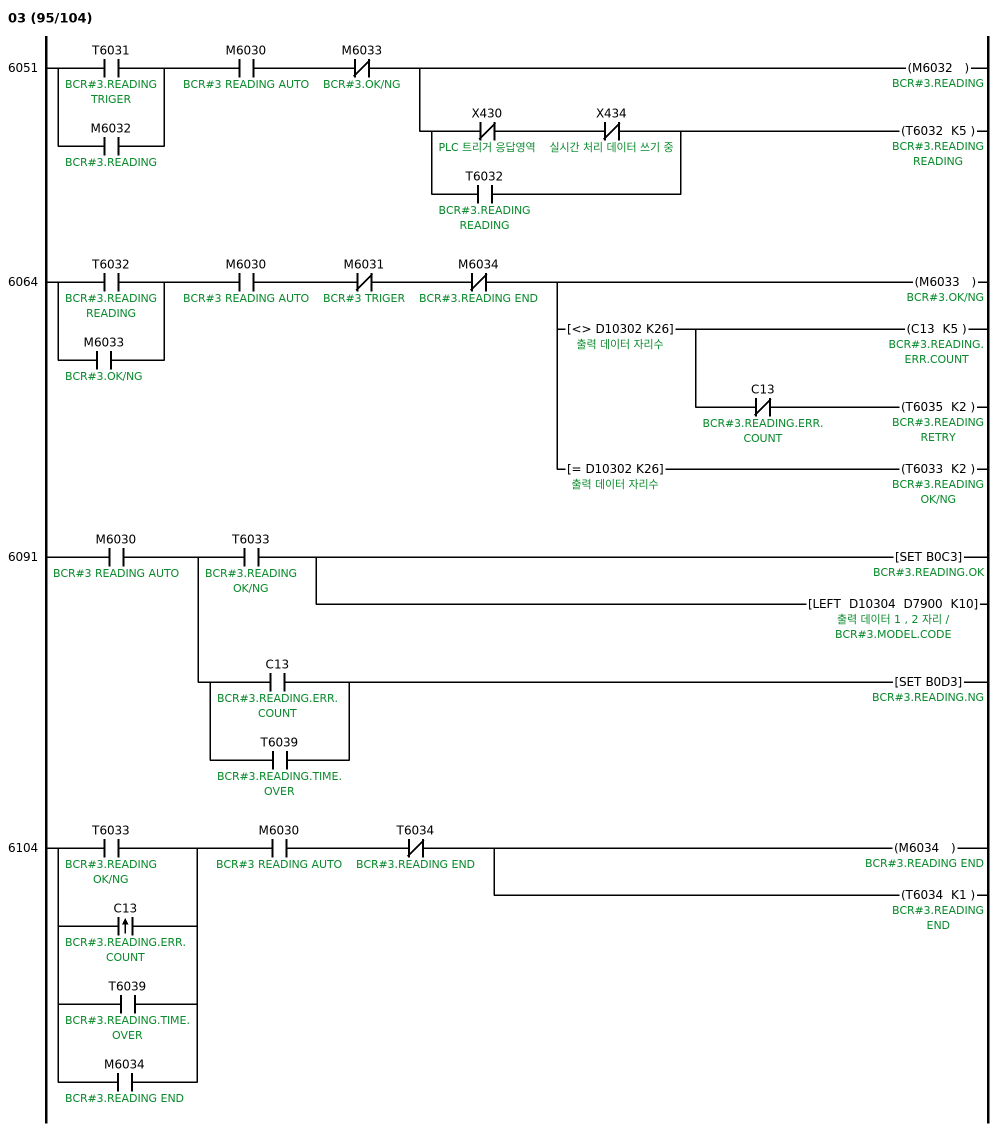
6051  LD      T6031  ; BCR#3.READING TRIGER
      OR      M6032  ; BCR#3.READING
      AND     M6030  ; BCR#3 READING AUTO
      ANI     M6033  ; BCR#3.OK/NG
      OUT     M6032  ; BCR#3.READING
      LDI     X430  ; PLC 트리거 응답영역
      ANI     X434  ; 실시간 처리 데이터 쓰기 중
      OR      T6032  ; BCR#3.READING READING
      ANB
      OUT     T6032 K5  ; BCR#3.READING READING
6064  LD      T6032  ; BCR#3.READING READING
      OR      M6033  ; BCR#3.OK/NG
      AND     M6030  ; BCR#3 READING AUTO
      ANI     M6031  ; BCR#3 TRIGER
      ANI     M6034  ; BCR#3.READING END
      OUT     M6033  ; BCR#3.OK/NG
      MPS
      AND<>   D10302 K26  ; 출력 데이터 자리수
      OUT     C13 K5  ; BCR#3.READING.ERR.COUNT
      ANI     C13  ; BCR#3.READING.ERR.COUNT
      OUT     T6035 K2  ; BCR#3.READING RETRY
      MPP
      AND=    D10302 K26  ; 출력 데이터 자리수
      OUT     T6033 K2  ; BCR#3.READING OK/NG
6091  LD      M6030  ; BCR#3 READING AUTO
      MPS
      AND     T6033  ; BCR#3.READING OK/NG
      SET     B0C3  ; BCR#3.READING.OK
      LEFT    D10304 D7900 K10  ; BCR#3.MODEL.CODE
      MPP
      LD      C13  ; BCR#3.READING.ERR.COUNT
      OR      T6039  ; BCR#3.READING.TIME.OVER
      ANB
      SET     B0D3  ; BCR#3.READING.NG
6104  LD      T6033  ; BCR#3.READING OK/NG
      ORP     C13  ; BCR#3.READING.ERR.COUNT
      OR      T6039  ; BCR#3.READING.TIME.OVER
      OR      M6034  ; BCR#3.READING END
      AND     M6030  ; BCR#3 READING AUTO
      ANI     T6034  ; BCR#3.READING END
      OUT     M6034  ; BCR#3.READING END
      OUT     T6034 K1  ; BCR#3.READING END
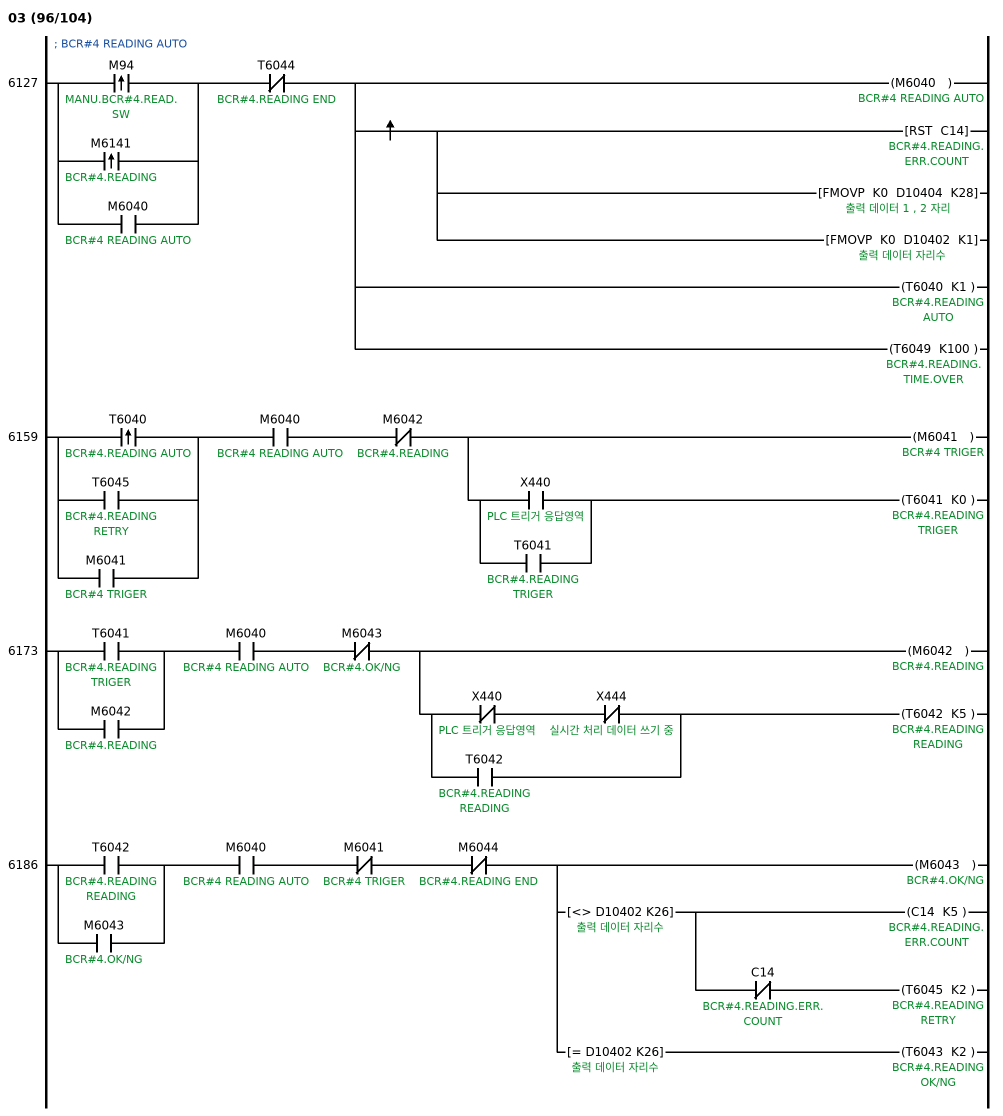
; BCR#4 READING AUTO
6127  LDP     M94  ; MANU.BCR#4.READ.SW
      ORP     M6141  ; BCR#4.READING
      OR      M6040  ; BCR#4 READING AUTO
      ANI     T6044  ; BCR#4.READING END
      OUT     M6040  ; BCR#4 READING AUTO
      MPS
      MEP
      RST     C14  ; BCR#4.READING.ERR.COUNT
      FMOVP   K0 D10404 K28  ; 출력 데이터 1 , 2 자리
      FMOVP   K0 D10402 K1  ; 출력 데이터 자리수
      MPP
      OUT     T6040 K1  ; BCR#4.READING AUTO
      OUT     T6049 K100  ; BCR#4.READING.TIME.OVER
6159  LDP     T6040  ; BCR#4.READING AUTO
      OR      T6045  ; BCR#4.READING RETRY
      OR      M6041  ; BCR#4 TRIGER
      AND     M6040  ; BCR#4 READING AUTO
      ANI     M6042  ; BCR#4.READING
      OUT     M6041  ; BCR#4 TRIGER
      LD      X440  ; PLC 트리거 응답영역
      OR      T6041  ; BCR#4.READING TRIGER
      ANB
      OUT     T6041 K0  ; BCR#4.READING TRIGER
6173  LD      T6041  ; BCR#4.READING TRIGER
      OR      M6042  ; BCR#4.READING
      AND     M6040  ; BCR#4 READING AUTO
      ANI     M6043  ; BCR#4.OK/NG
      OUT     M6042  ; BCR#4.READING
      LDI     X440  ; PLC 트리거 응답영역
      ANI     X444  ; 실시간 처리 데이터 쓰기 중
      OR      T6042  ; BCR#4.READING READING
      ANB
      OUT     T6042 K5  ; BCR#4.READING READING
6186  LD      T6042  ; BCR#4.READING READING
      OR      M6043  ; BCR#4.OK/NG
      AND     M6040  ; BCR#4 READING AUTO
      ANI     M6041  ; BCR#4 TRIGER
      ANI     M6044  ; BCR#4.READING END
      OUT     M6043  ; BCR#4.OK/NG
      MPS
      AND<>   D10402 K26  ; 출력 데이터 자리수
      OUT     C14 K5  ; BCR#4.READING.ERR.COUNT
      ANI     C14  ; BCR#4.READING.ERR.COUNT
      OUT     T6045 K2  ; BCR#4.READING RETRY
      MPP
      AND=    D10402 K26  ; 출력 데이터 자리수
      OUT     T6043 K2  ; BCR#4.READING OK/NG
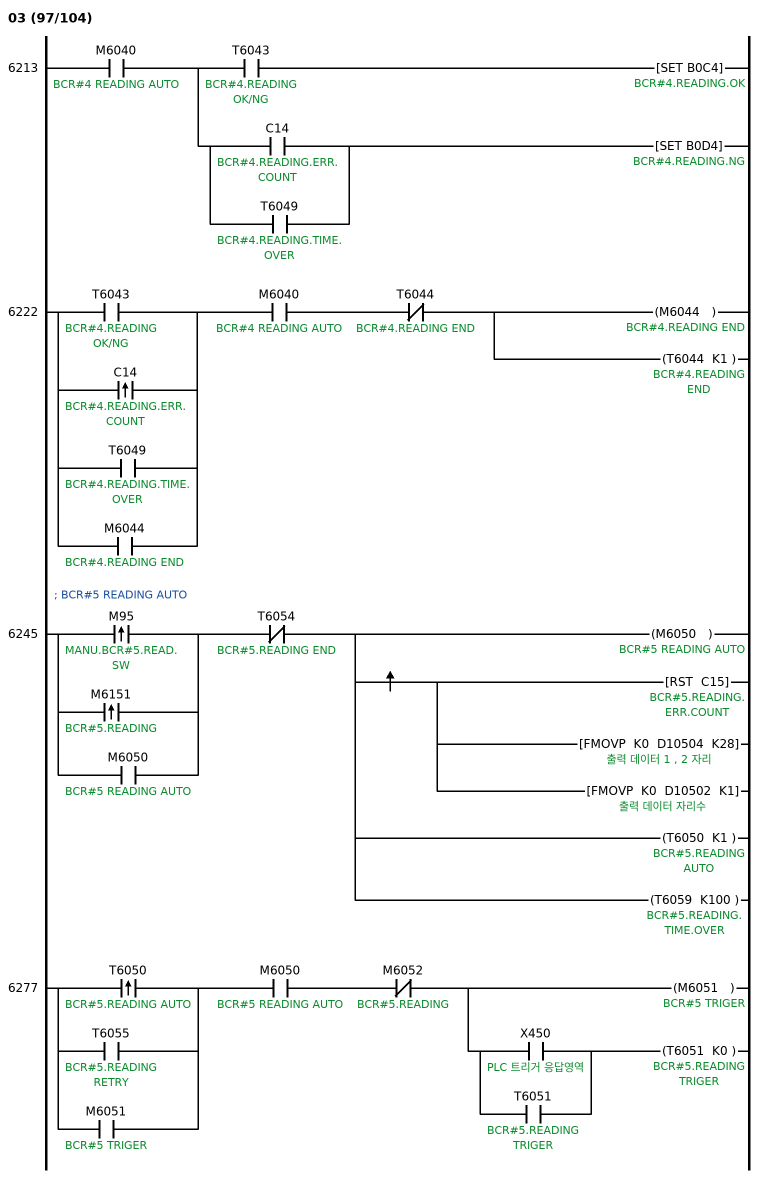
6213  LD      M6040  ; BCR#4 READING AUTO
      MPS
      AND     T6043  ; BCR#4.READING OK/NG
      SET     B0C4  ; BCR#4.READING.OK
      MPP
      LD      C14  ; BCR#4.READING.ERR.COUNT
      OR      T6049  ; BCR#4.READING.TIME.OVER
      ANB
      SET     B0D4  ; BCR#4.READING.NG
6222  LD      T6043  ; BCR#4.READING OK/NG
      ORP     C14  ; BCR#4.READING.ERR.COUNT
      OR      T6049  ; BCR#4.READING.TIME.OVER
      OR      M6044  ; BCR#4.READING END
      AND     M6040  ; BCR#4 READING AUTO
      ANI     T6044  ; BCR#4.READING END
      OUT     M6044  ; BCR#4.READING END
      OUT     T6044 K1  ; BCR#4.READING END
; BCR#5 READING AUTO
6245  LDP     M95  ; MANU.BCR#5.READ.SW
      ORP     M6151  ; BCR#5.READING
      OR      M6050  ; BCR#5 READING AUTO
      ANI     T6054  ; BCR#5.READING END
      OUT     M6050  ; BCR#5 READING AUTO
      MPS
      MEP
      RST     C15  ; BCR#5.READING.ERR.COUNT
      FMOVP   K0 D10504 K28  ; 출력 데이터 1 , 2 자리
      FMOVP   K0 D10502 K1  ; 출력 데이터 자리수
      MPP
      OUT     T6050 K1  ; BCR#5.READING AUTO
      OUT     T6059 K100  ; BCR#5.READING.TIME.OVER
6277  LDP     T6050  ; BCR#5.READING AUTO
      OR      T6055  ; BCR#5.READING RETRY
      OR      M6051  ; BCR#5 TRIGER
      AND     M6050  ; BCR#5 READING AUTO
      ANI     M6052  ; BCR#5.READING
      OUT     M6051  ; BCR#5 TRIGER
      LD      X450  ; PLC 트리거 응답영역
      OR      T6051  ; BCR#5.READING TRIGER
      ANB
      OUT     T6051 K0  ; BCR#5.READING TRIGER
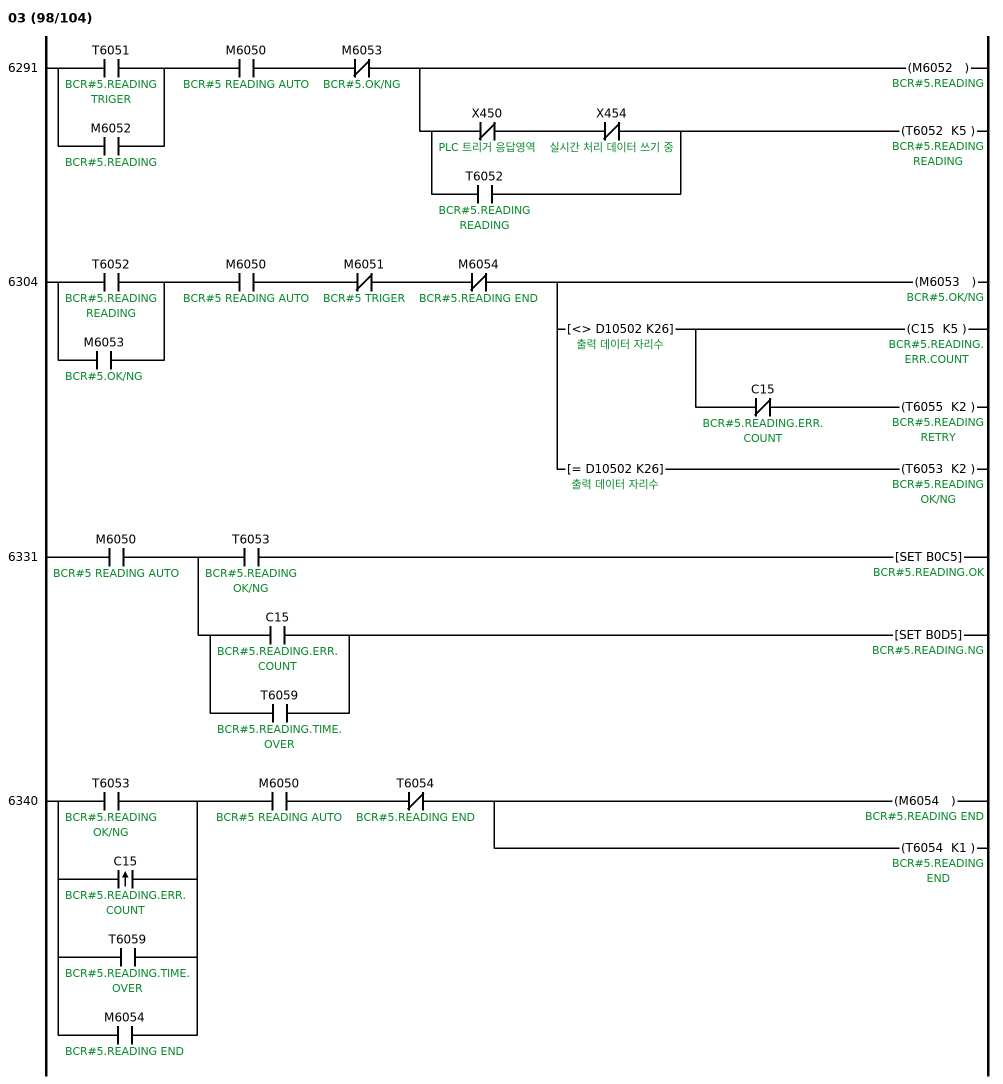
6291  LD      T6051  ; BCR#5.READING TRIGER
      OR      M6052  ; BCR#5.READING
      AND     M6050  ; BCR#5 READING AUTO
      ANI     M6053  ; BCR#5.OK/NG
      OUT     M6052  ; BCR#5.READING
      LDI     X450  ; PLC 트리거 응답영역
      ANI     X454  ; 실시간 처리 데이터 쓰기 중
      OR      T6052  ; BCR#5.READING READING
      ANB
      OUT     T6052 K5  ; BCR#5.READING READING
6304  LD      T6052  ; BCR#5.READING READING
      OR      M6053  ; BCR#5.OK/NG
      AND     M6050  ; BCR#5 READING AUTO
      ANI     M6051  ; BCR#5 TRIGER
      ANI     M6054  ; BCR#5.READING END
      OUT     M6053  ; BCR#5.OK/NG
      MPS
      AND<>   D10502 K26  ; 출력 데이터 자리수
      OUT     C15 K5  ; BCR#5.READING.ERR.COUNT
      ANI     C15  ; BCR#5.READING.ERR.COUNT
      OUT     T6055 K2  ; BCR#5.READING RETRY
      MPP
      AND=    D10502 K26  ; 출력 데이터 자리수
      OUT     T6053 K2  ; BCR#5.READING OK/NG
6331  LD      M6050  ; BCR#5 READING AUTO
      MPS
      AND     T6053  ; BCR#5.READING OK/NG
      SET     B0C5  ; BCR#5.READING.OK
      MPP
      LD      C15  ; BCR#5.READING.ERR.COUNT
      OR      T6059  ; BCR#5.READING.TIME.OVER
      ANB
      SET     B0D5  ; BCR#5.READING.NG
6340  LD      T6053  ; BCR#5.READING OK/NG
      ORP     C15  ; BCR#5.READING.ERR.COUNT
      OR      T6059  ; BCR#5.READING.TIME.OVER
      OR      M6054  ; BCR#5.READING END
      AND     M6050  ; BCR#5 READING AUTO
      ANI     T6054  ; BCR#5.READING END
      OUT     M6054  ; BCR#5.READING END
      OUT     T6054 K1  ; BCR#5.READING END
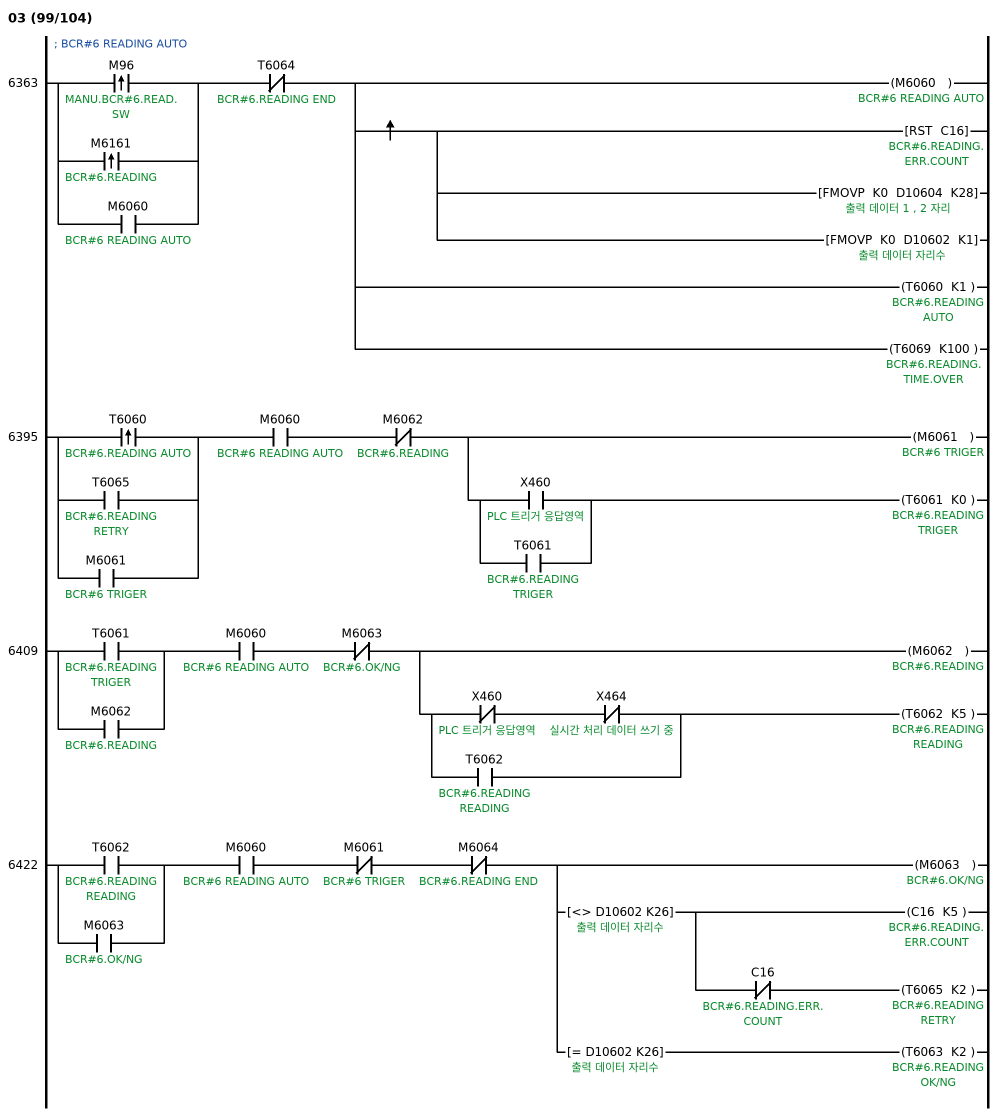
; BCR#6 READING AUTO
6363  LDP     M96  ; MANU.BCR#6.READ.SW
      ORP     M6161  ; BCR#6.READING
      OR      M6060  ; BCR#6 READING AUTO
      ANI     T6064  ; BCR#6.READING END
      OUT     M6060  ; BCR#6 READING AUTO
      MPS
      MEP
      RST     C16  ; BCR#6.READING.ERR.COUNT
      FMOVP   K0 D10604 K28  ; 출력 데이터 1 , 2 자리
      FMOVP   K0 D10602 K1  ; 출력 데이터 자리수
      MPP
      OUT     T6060 K1  ; BCR#6.READING AUTO
      OUT     T6069 K100  ; BCR#6.READING.TIME.OVER
6395  LDP     T6060  ; BCR#6.READING AUTO
      OR      T6065  ; BCR#6.READING RETRY
      OR      M6061  ; BCR#6 TRIGER
      AND     M6060  ; BCR#6 READING AUTO
      ANI     M6062  ; BCR#6.READING
      OUT     M6061  ; BCR#6 TRIGER
      LD      X460  ; PLC 트리거 응답영역
      OR      T6061  ; BCR#6.READING TRIGER
      ANB
      OUT     T6061 K0  ; BCR#6.READING TRIGER
6409  LD      T6061  ; BCR#6.READING TRIGER
      OR      M6062  ; BCR#6.READING
      AND     M6060  ; BCR#6 READING AUTO
      ANI     M6063  ; BCR#6.OK/NG
      OUT     M6062  ; BCR#6.READING
      LDI     X460  ; PLC 트리거 응답영역
      ANI     X464  ; 실시간 처리 데이터 쓰기 중
      OR      T6062  ; BCR#6.READING READING
      ANB
      OUT     T6062 K5  ; BCR#6.READING READING
6422  LD      T6062  ; BCR#6.READING READING
      OR      M6063  ; BCR#6.OK/NG
      AND     M6060  ; BCR#6 READING AUTO
      ANI     M6061  ; BCR#6 TRIGER
      ANI     M6064  ; BCR#6.READING END
      OUT     M6063  ; BCR#6.OK/NG
      MPS
      AND<>   D10602 K26  ; 출력 데이터 자리수
      OUT     C16 K5  ; BCR#6.READING.ERR.COUNT
      ANI     C16  ; BCR#6.READING.ERR.COUNT
      OUT     T6065 K2  ; BCR#6.READING RETRY
      MPP
      AND=    D10602 K26  ; 출력 데이터 자리수
      OUT     T6063 K2  ; BCR#6.READING OK/NG
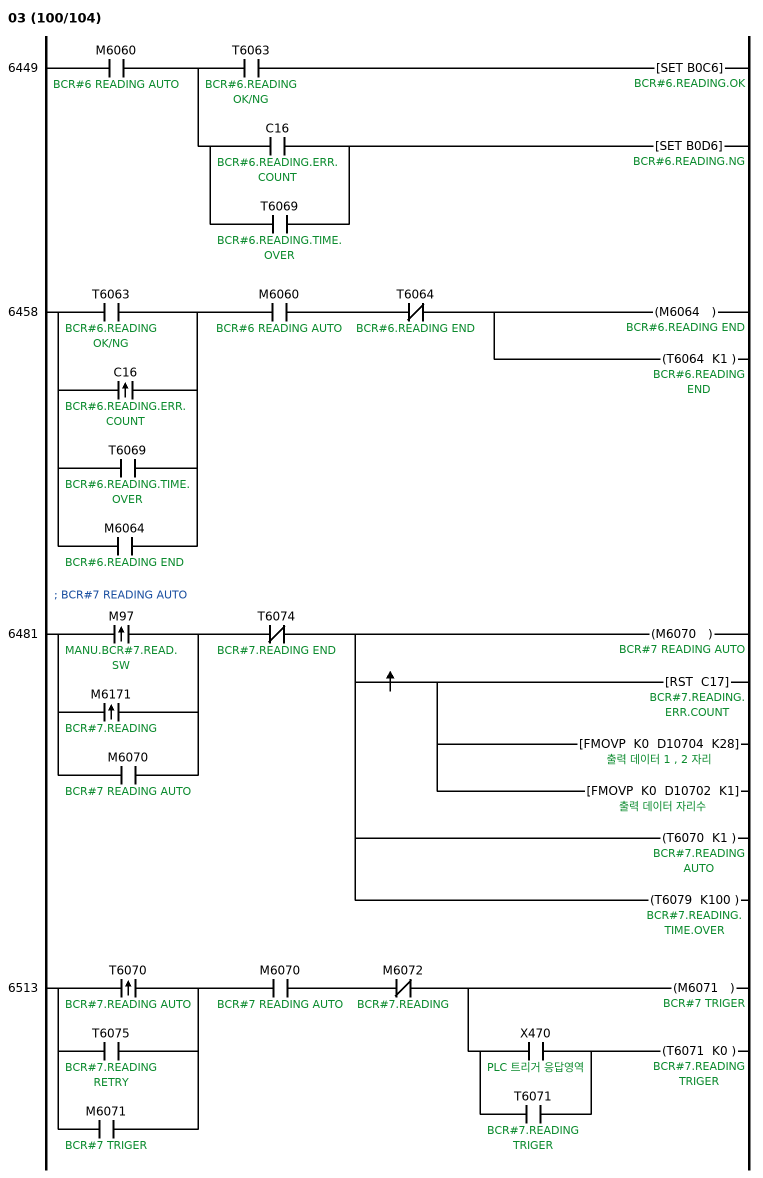
6449  LD      M6060  ; BCR#6 READING AUTO
      MPS
      AND     T6063  ; BCR#6.READING OK/NG
      SET     B0C6  ; BCR#6.READING.OK
      MPP
      LD      C16  ; BCR#6.READING.ERR.COUNT
      OR      T6069  ; BCR#6.READING.TIME.OVER
      ANB
      SET     B0D6  ; BCR#6.READING.NG
6458  LD      T6063  ; BCR#6.READING OK/NG
      ORP     C16  ; BCR#6.READING.ERR.COUNT
      OR      T6069  ; BCR#6.READING.TIME.OVER
      OR      M6064  ; BCR#6.READING END
      AND     M6060  ; BCR#6 READING AUTO
      ANI     T6064  ; BCR#6.READING END
      OUT     M6064  ; BCR#6.READING END
      OUT     T6064 K1  ; BCR#6.READING END
; BCR#7 READING AUTO
6481  LDP     M97  ; MANU.BCR#7.READ.SW
      ORP     M6171  ; BCR#7.READING
      OR      M6070  ; BCR#7 READING AUTO
      ANI     T6074  ; BCR#7.READING END
      OUT     M6070  ; BCR#7 READING AUTO
      MPS
      MEP
      RST     C17  ; BCR#7.READING.ERR.COUNT
      FMOVP   K0 D10704 K28  ; 출력 데이터 1 , 2 자리
      FMOVP   K0 D10702 K1  ; 출력 데이터 자리수
      MPP
      OUT     T6070 K1  ; BCR#7.READING AUTO
      OUT     T6079 K100  ; BCR#7.READING.TIME.OVER
6513  LDP     T6070  ; BCR#7.READING AUTO
      OR      T6075  ; BCR#7.READING RETRY
      OR      M6071  ; BCR#7 TRIGER
      AND     M6070  ; BCR#7 READING AUTO
      ANI     M6072  ; BCR#7.READING
      OUT     M6071  ; BCR#7 TRIGER
      LD      X470  ; PLC 트리거 응답영역
      OR      T6071  ; BCR#7.READING TRIGER
      ANB
      OUT     T6071 K0  ; BCR#7.READING TRIGER
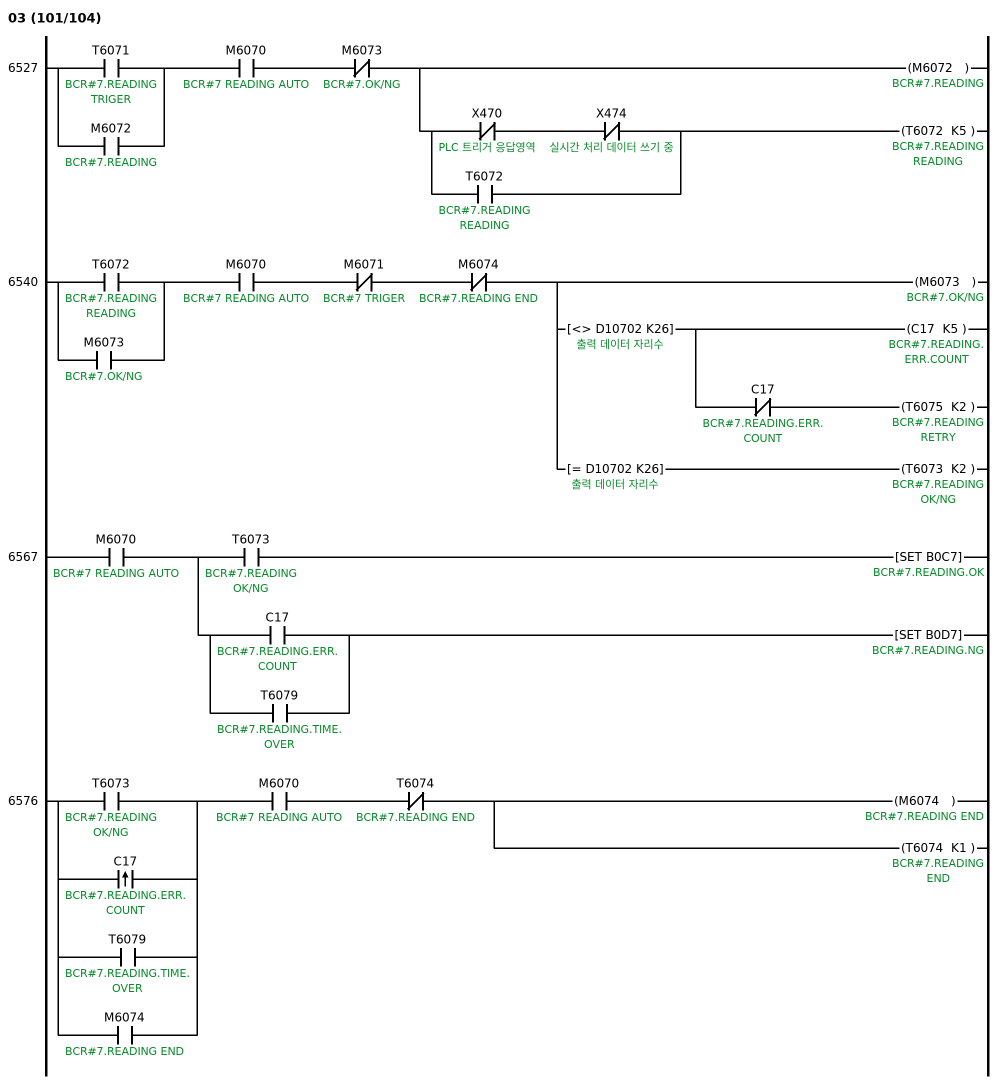
6527  LD      T6071  ; BCR#7.READING TRIGER
      OR      M6072  ; BCR#7.READING
      AND     M6070  ; BCR#7 READING AUTO
      ANI     M6073  ; BCR#7.OK/NG
      OUT     M6072  ; BCR#7.READING
      LDI     X470  ; PLC 트리거 응답영역
      ANI     X474  ; 실시간 처리 데이터 쓰기 중
      OR      T6072  ; BCR#7.READING READING
      ANB
      OUT     T6072 K5  ; BCR#7.READING READING
6540  LD      T6072  ; BCR#7.READING READING
      OR      M6073  ; BCR#7.OK/NG
      AND     M6070  ; BCR#7 READING AUTO
      ANI     M6071  ; BCR#7 TRIGER
      ANI     M6074  ; BCR#7.READING END
      OUT     M6073  ; BCR#7.OK/NG
      MPS
      AND<>   D10702 K26  ; 출력 데이터 자리수
      OUT     C17 K5  ; BCR#7.READING.ERR.COUNT
      ANI     C17  ; BCR#7.READING.ERR.COUNT
      OUT     T6075 K2  ; BCR#7.READING RETRY
      MPP
      AND=    D10702 K26  ; 출력 데이터 자리수
      OUT     T6073 K2  ; BCR#7.READING OK/NG
6567  LD      M6070  ; BCR#7 READING AUTO
      MPS
      AND     T6073  ; BCR#7.READING OK/NG
      SET     B0C7  ; BCR#7.READING.OK
      MPP
      LD      C17  ; BCR#7.READING.ERR.COUNT
      OR      T6079  ; BCR#7.READING.TIME.OVER
      ANB
      SET     B0D7  ; BCR#7.READING.NG
6576  LD      T6073  ; BCR#7.READING OK/NG
      ORP     C17  ; BCR#7.READING.ERR.COUNT
      OR      T6079  ; BCR#7.READING.TIME.OVER
      OR      M6074  ; BCR#7.READING END
      AND     M6070  ; BCR#7 READING AUTO
      ANI     T6074  ; BCR#7.READING END
      OUT     M6074  ; BCR#7.READING END
      OUT     T6074 K1  ; BCR#7.READING END
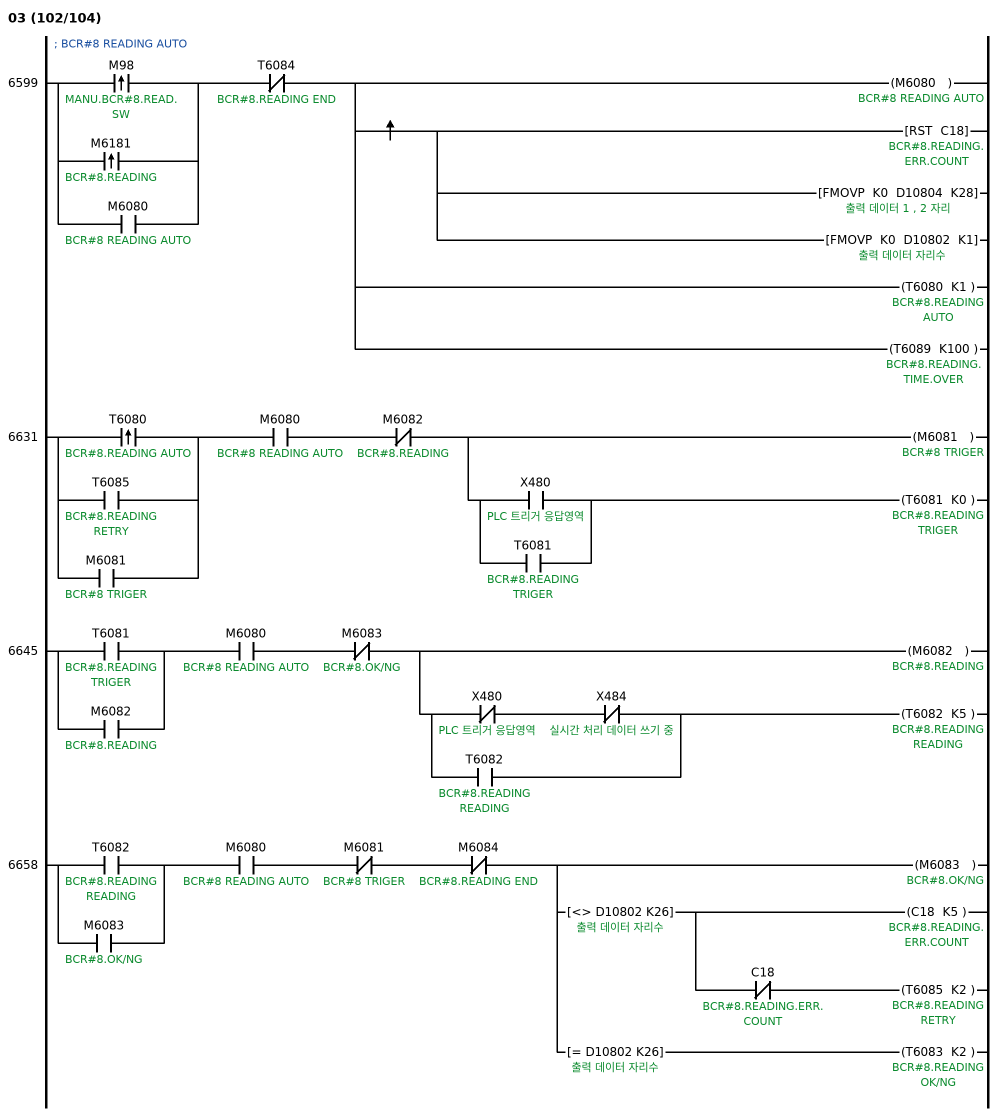
; BCR#8 READING AUTO
6599  LDP     M98  ; MANU.BCR#8.READ.SW
      ORP     M6181  ; BCR#8.READING
      OR      M6080  ; BCR#8 READING AUTO
      ANI     T6084  ; BCR#8.READING END
      OUT     M6080  ; BCR#8 READING AUTO
      MPS
      MEP
      RST     C18  ; BCR#8.READING.ERR.COUNT
      FMOVP   K0 D10804 K28  ; 출력 데이터 1 , 2 자리
      FMOVP   K0 D10802 K1  ; 출력 데이터 자리수
      MPP
      OUT     T6080 K1  ; BCR#8.READING AUTO
      OUT     T6089 K100  ; BCR#8.READING.TIME.OVER
6631  LDP     T6080  ; BCR#8.READING AUTO
      OR      T6085  ; BCR#8.READING RETRY
      OR      M6081  ; BCR#8 TRIGER
      AND     M6080  ; BCR#8 READING AUTO
      ANI     M6082  ; BCR#8.READING
      OUT     M6081  ; BCR#8 TRIGER
      LD      X480  ; PLC 트리거 응답영역
      OR      T6081  ; BCR#8.READING TRIGER
      ANB
      OUT     T6081 K0  ; BCR#8.READING TRIGER
6645  LD      T6081  ; BCR#8.READING TRIGER
      OR      M6082  ; BCR#8.READING
      AND     M6080  ; BCR#8 READING AUTO
      ANI     M6083  ; BCR#8.OK/NG
      OUT     M6082  ; BCR#8.READING
      LDI     X480  ; PLC 트리거 응답영역
      ANI     X484  ; 실시간 처리 데이터 쓰기 중
      OR      T6082  ; BCR#8.READING READING
      ANB
      OUT     T6082 K5  ; BCR#8.READING READING
6658  LD      T6082  ; BCR#8.READING READING
      OR      M6083  ; BCR#8.OK/NG
      AND     M6080  ; BCR#8 READING AUTO
      ANI     M6081  ; BCR#8 TRIGER
      ANI     M6084  ; BCR#8.READING END
      OUT     M6083  ; BCR#8.OK/NG
      MPS
      AND<>   D10802 K26  ; 출력 데이터 자리수
      OUT     C18 K5  ; BCR#8.READING.ERR.COUNT
      ANI     C18  ; BCR#8.READING.ERR.COUNT
      OUT     T6085 K2  ; BCR#8.READING RETRY
      MPP
      AND=    D10802 K26  ; 출력 데이터 자리수
      OUT     T6083 K2  ; BCR#8.READING OK/NG
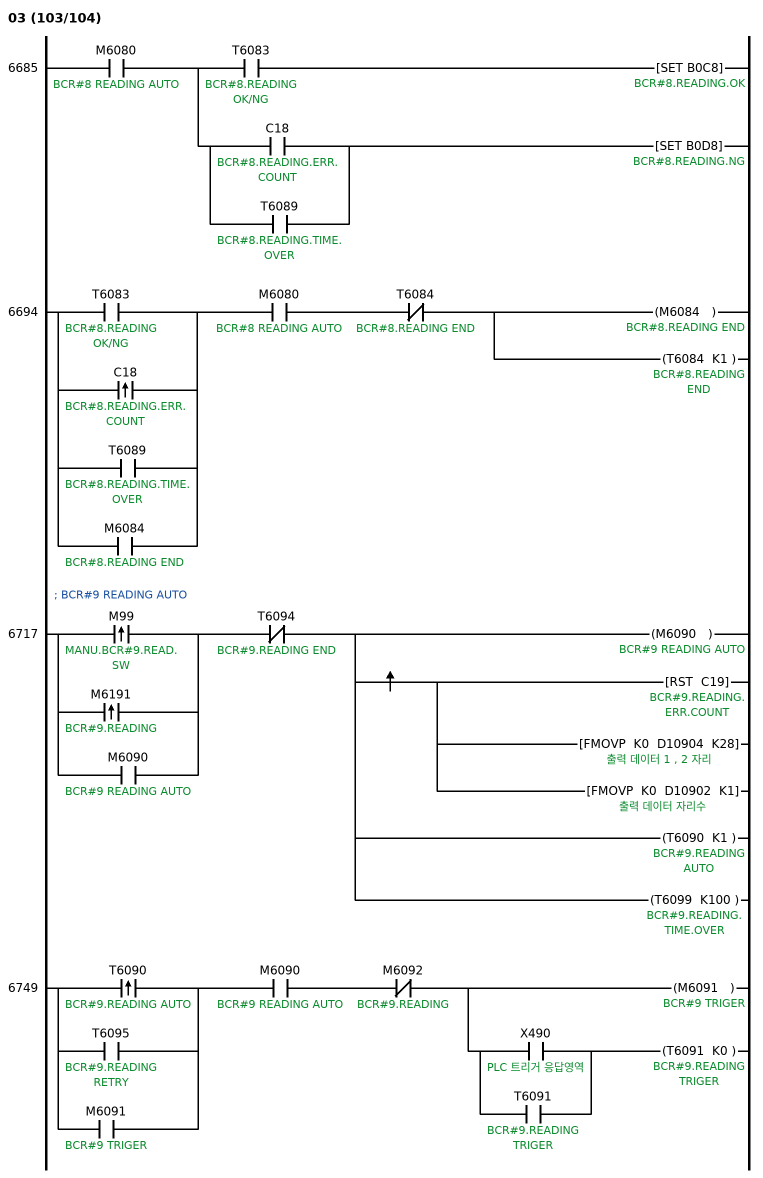
6685  LD      M6080  ; BCR#8 READING AUTO
      MPS
      AND     T6083  ; BCR#8.READING OK/NG
      SET     B0C8  ; BCR#8.READING.OK
      MPP
      LD      C18  ; BCR#8.READING.ERR.COUNT
      OR      T6089  ; BCR#8.READING.TIME.OVER
      ANB
      SET     B0D8  ; BCR#8.READING.NG
6694  LD      T6083  ; BCR#8.READING OK/NG
      ORP     C18  ; BCR#8.READING.ERR.COUNT
      OR      T6089  ; BCR#8.READING.TIME.OVER
      OR      M6084  ; BCR#8.READING END
      AND     M6080  ; BCR#8 READING AUTO
      ANI     T6084  ; BCR#8.READING END
      OUT     M6084  ; BCR#8.READING END
      OUT     T6084 K1  ; BCR#8.READING END
; BCR#9 READING AUTO
6717  LDP     M99  ; MANU.BCR#9.READ.SW
      ORP     M6191  ; BCR#9.READING
      OR      M6090  ; BCR#9 READING AUTO
      ANI     T6094  ; BCR#9.READING END
      OUT     M6090  ; BCR#9 READING AUTO
      MPS
      MEP
      RST     C19  ; BCR#9.READING.ERR.COUNT
      FMOVP   K0 D10904 K28  ; 출력 데이터 1 , 2 자리
      FMOVP   K0 D10902 K1  ; 출력 데이터 자리수
      MPP
      OUT     T6090 K1  ; BCR#9.READING AUTO
      OUT     T6099 K100  ; BCR#9.READING.TIME.OVER
6749  LDP     T6090  ; BCR#9.READING AUTO
      OR      T6095  ; BCR#9.READING RETRY
      OR      M6091  ; BCR#9 TRIGER
      AND     M6090  ; BCR#9 READING AUTO
      ANI     M6092  ; BCR#9.READING
      OUT     M6091  ; BCR#9 TRIGER
      LD      X490  ; PLC 트리거 응답영역
      OR      T6091  ; BCR#9.READING TRIGER
      ANB
      OUT     T6091 K0  ; BCR#9.READING TRIGER
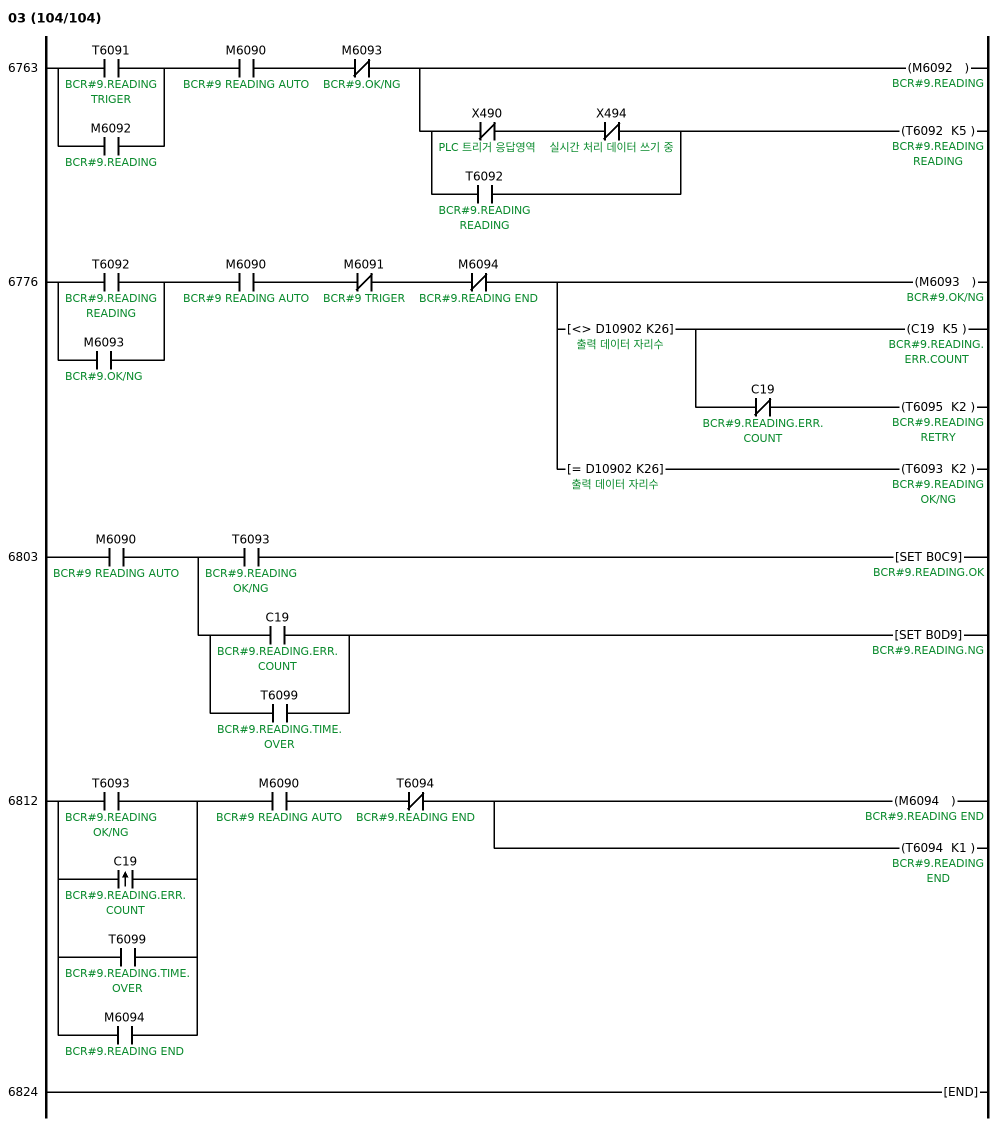
6763  LD      T6091  ; BCR#9.READING TRIGER
      OR      M6092  ; BCR#9.READING
      AND     M6090  ; BCR#9 READING AUTO
      ANI     M6093  ; BCR#9.OK/NG
      OUT     M6092  ; BCR#9.READING
      LDI     X490  ; PLC 트리거 응답영역
      ANI     X494  ; 실시간 처리 데이터 쓰기 중
      OR      T6092  ; BCR#9.READING READING
      ANB
      OUT     T6092 K5  ; BCR#9.READING READING
6776  LD      T6092  ; BCR#9.READING READING
      OR      M6093  ; BCR#9.OK/NG
      AND     M6090  ; BCR#9 READING AUTO
      ANI     M6091  ; BCR#9 TRIGER
      ANI     M6094  ; BCR#9.READING END
      OUT     M6093  ; BCR#9.OK/NG
      MPS
      AND<>   D10902 K26  ; 출력 데이터 자리수
      OUT     C19 K5  ; BCR#9.READING.ERR.COUNT
      ANI     C19  ; BCR#9.READING.ERR.COUNT
      OUT     T6095 K2  ; BCR#9.READING RETRY
      MPP
      AND=    D10902 K26  ; 출력 데이터 자리수
      OUT     T6093 K2  ; BCR#9.READING OK/NG
6803  LD      M6090  ; BCR#9 READING AUTO
      MPS
      AND     T6093  ; BCR#9.READING OK/NG
      SET     B0C9  ; BCR#9.READING.OK
      MPP
      LD      C19  ; BCR#9.READING.ERR.COUNT
      OR      T6099  ; BCR#9.READING.TIME.OVER
      ANB
      SET     B0D9  ; BCR#9.READING.NG
6812  LD      T6093  ; BCR#9.READING OK/NG
      ORP     C19  ; BCR#9.READING.ERR.COUNT
      OR      T6099  ; BCR#9.READING.TIME.OVER
      OR      M6094  ; BCR#9.READING END
      AND     M6090  ; BCR#9 READING AUTO
      ANI     T6094  ; BCR#9.READING END
      OUT     M6094  ; BCR#9.READING END
      OUT     T6094 K1  ; BCR#9.READING END
6824  END
END_PROGRAM

PROGRAM 04  // SERVO
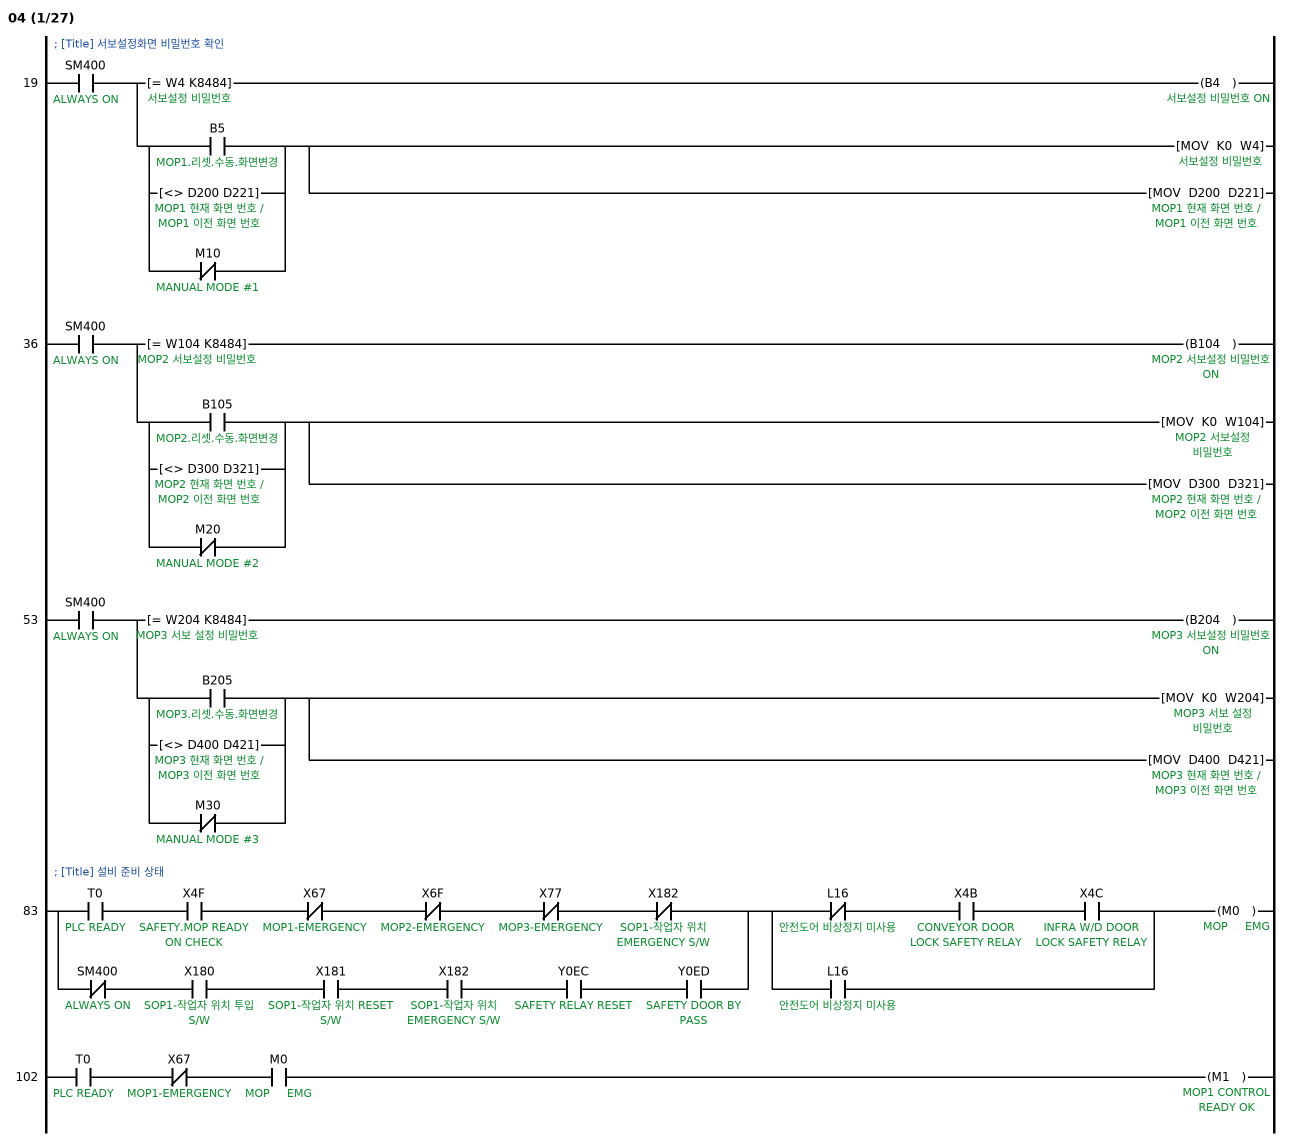
; [Title] 서보설정화면 비밀번호 확인
19    LD      SM400  ; ALWAYS ON
      MPS
      AND=    W4 K8484  ; 서보설정 비밀번호
      OUT     B4  ; 서보설정 비밀번호 ON
      MPP
      LD      B5  ; MOP1.리셋.수동.화면변경
      OR<>    D200 D221  ; MOP1 현재 화면 번호 / MOP1 이전 화면 번호
      ORI     M10  ; MANUAL MODE #1
      ANB
      MOV     K0 W4
      MOV     D200 D221
36    LD      SM400  ; ALWAYS ON
      MPS
      AND=    W104 K8484  ; MOP2 서보설정 비밀번호
      OUT     B104  ; MOP2 서보설정 비밀번호 ON
      MPP
      LD      B105  ; MOP2.리셋.수동.화면변경
      OR<>    D300 D321  ; MOP2 현재 화면 번호 / MOP2 이전 화면 번호
      ORI     M20  ; MANUAL MODE #2
      ANB
      MOV     K0 W104
      MOV     D300 D321
53    LD      SM400  ; ALWAYS ON
      MPS
      AND=    W204 K8484  ; MOP3 서보 설정 비밀번호
      OUT     B204  ; MOP3 서보설정 비밀번호 ON
      MPP
      LD      B205  ; MOP3.리셋.수동.화면변경
      OR<>    D400 D421  ; MOP3 현재 화면 번호 / MOP3 이전 화면 번호
      ORI     M30  ; MANUAL MODE #3
      ANB
      MOV     K0 W204
      MOV     D400 D421
; [Title] 설비 준비 상태
83    LD      T0  ; PLC READY
      AND     X4F  ; SAFETY.MOP READY ON CHECK
      ANI     X67  ; MOP1-EMERGENCY
      ANI     X6F  ; MOP2-EMERGENCY
      ANI     X77  ; MOP3-EMERGENCY
      ANI     X182  ; SOP1-작업자 위치 EMERGENCY S/W
      LDI     SM400  ; ALWAYS ON
      AND     X180  ; SOP1-작업자 위치 투입 S/W
      AND     X181  ; SOP1-작업자 위치 RESET S/W
      AND     X182  ; SOP1-작업자 위치 EMERGENCY S/W
      AND     Y0EC  ; SAFETY RELAY RESET
      AND     Y0ED  ; SAFETY DOOR BY PASS
      ORB
      LDI     L16  ; 안전도어 비상정지 미사용
      AND     X4B  ; CONVEYOR DOOR LOCK SAFETY RELAY
      AND     X4C  ; INFRA W/D DOOR LOCK SAFETY RELAY
      OR      L16  ; 안전도어 비상정지 미사용
      ANB
      OUT     M0  ; MOP     EMG
102   LD      T0  ; PLC READY
      ANI     X67  ; MOP1-EMERGENCY
      AND     M0  ; MOP     EMG
      OUT     M1  ; MOP1 CONTROL READY OK
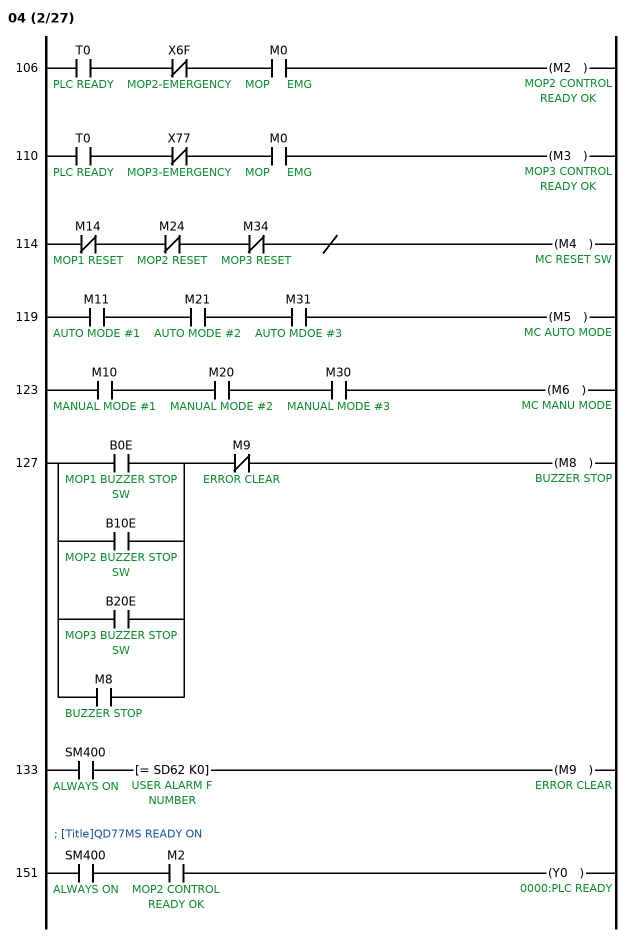
106   LD      T0  ; PLC READY
      ANI     X6F  ; MOP2-EMERGENCY
      AND     M0  ; MOP     EMG
      OUT     M2  ; MOP2 CONTROL READY OK
110   LD      T0  ; PLC READY
      ANI     X77  ; MOP3-EMERGENCY
      AND     M0  ; MOP     EMG
      OUT     M3  ; MOP3 CONTROL READY OK
114   LDI     M14  ; MOP1 RESET
      ANI     M24  ; MOP2 RESET
      ANI     M34  ; MOP3 RESET
      INV
      OUT     M4  ; MC RESET SW
119   LD      M11  ; AUTO MODE #1
      AND     M21  ; AUTO MODE #2
      AND     M31  ; AUTO MDOE #3
      OUT     M5  ; MC AUTO MODE
123   LD      M10  ; MANUAL MODE #1
      AND     M20  ; MANUAL MODE #2
      AND     M30  ; MANUAL MODE #3
      OUT     M6  ; MC MANU MODE
127   LD      B0E  ; MOP1 BUZZER STOP SW
      OR      B10E  ; MOP2 BUZZER STOP SW
      OR      B20E  ; MOP3 BUZZER STOP SW
      OR      M8  ; BUZZER STOP
      ANI     M9  ; ERROR CLEAR
      OUT     M8  ; BUZZER STOP
133   LD      SM400  ; ALWAYS ON
      AND=    SD62 K0  ; USER ALARM F NUMBER
      OUT     M9  ; ERROR CLEAR
; [Title]QD77MS READY ON
151   LD      SM400  ; ALWAYS ON
      AND     M2  ; MOP2 CONTROL READY OK
      OUT     Y0  ; 0000:PLC READY
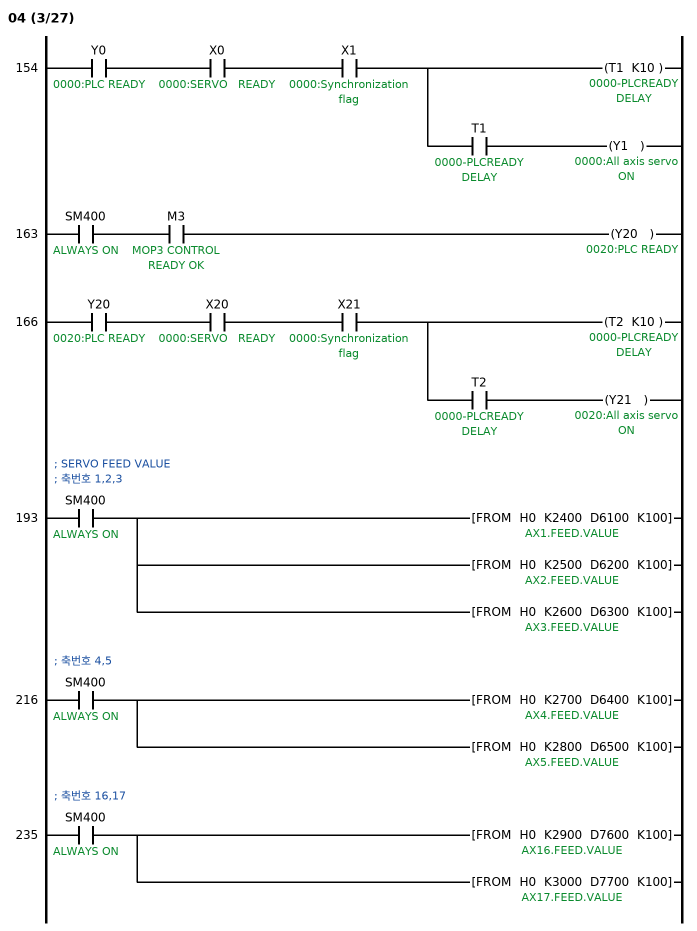
154   LD      Y0  ; 0000:PLC READY
      AND     X0  ; 0000:SERVO   READY
      AND     X1  ; 0000:Synchronization flag
      OUT     T1 K10  ; 0000-PLCREADY   DELAY
      AND     T1  ; 0000-PLCREADY   DELAY
      OUT     Y1  ; 0000:All axis servo  ON
163   LD      SM400  ; ALWAYS ON
      AND     M3  ; MOP3 CONTROL READY OK
      OUT     Y20  ; 0020:PLC READY
166   LD      Y20  ; 0020:PLC READY
      AND     X20  ; 0000:SERVO   READY
      AND     X21  ; 0000:Synchronization flag
      OUT     T2 K10  ; 0000-PLCREADY   DELAY
      AND     T2  ; 0000-PLCREADY   DELAY
      OUT     Y21  ; 0020:All axis servo  ON
; SERVO FEED VALUE
; 축번호 1,2,3
193   LD      SM400  ; ALWAYS ON
      FROM    H0 K2400 D6100 K100  ; AX1.FEED.VALUE
      FROM    H0 K2500 D6200 K100  ; AX2.FEED.VALUE
      FROM    H0 K2600 D6300 K100  ; AX3.FEED.VALUE
; 축번호 4,5
216   LD      SM400  ; ALWAYS ON
      FROM    H0 K2700 D6400 K100  ; AX4.FEED.VALUE
      FROM    H0 K2800 D6500 K100  ; AX5.FEED.VALUE
; 축번호 16,17
235   LD      SM400  ; ALWAYS ON
      FROM    H0 K2900 D7600 K100  ; AX16.FEED.VALUE
      FROM    H0 K3000 D7700 K100  ; AX17.FEED.VALUE
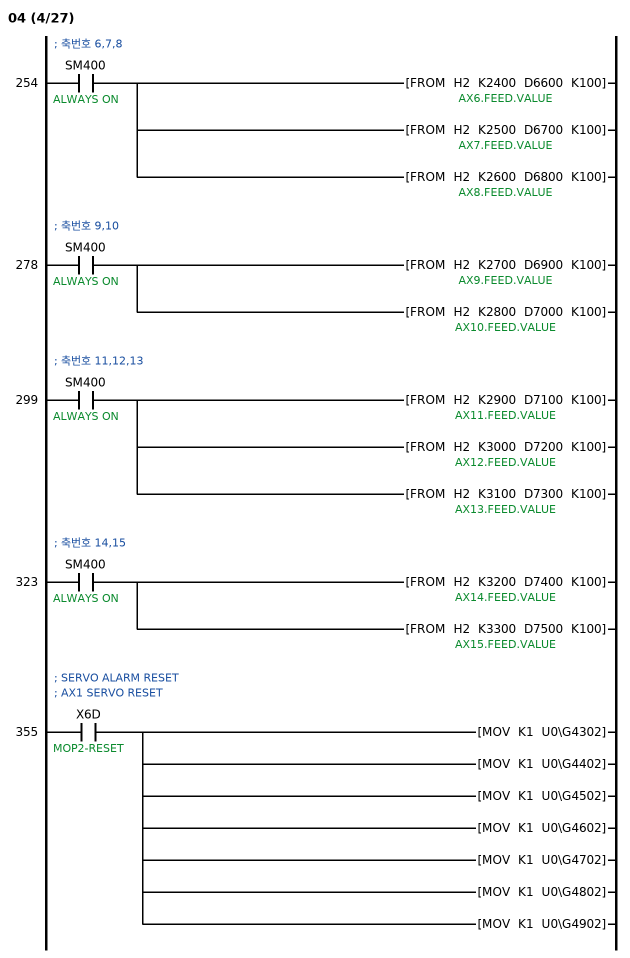
; 축번호 6,7,8
254   LD      SM400  ; ALWAYS ON
      FROM    H2 K2400 D6600 K100  ; AX6.FEED.VALUE
      FROM    H2 K2500 D6700 K100  ; AX7.FEED.VALUE
      FROM    H2 K2600 D6800 K100  ; AX8.FEED.VALUE
; 축번호 9,10
278   LD      SM400  ; ALWAYS ON
      FROM    H2 K2700 D6900 K100  ; AX9.FEED.VALUE
      FROM    H2 K2800 D7000 K100  ; AX10.FEED.VALUE
; 축번호 11,12,13
299   LD      SM400  ; ALWAYS ON
      FROM    H2 K2900 D7100 K100  ; AX11.FEED.VALUE
      FROM    H2 K3000 D7200 K100  ; AX12.FEED.VALUE
      FROM    H2 K3100 D7300 K100  ; AX13.FEED.VALUE
; 축번호 14,15
323   LD      SM400  ; ALWAYS ON
      FROM    H2 K3200 D7400 K100  ; AX14.FEED.VALUE
      FROM    H2 K3300 D7500 K100  ; AX15.FEED.VALUE
; SERVO ALARM RESET
; AX1 SERVO RESET
355   LD      X6D  ; MOP2-RESET
      MOV     K1 U0\G4302
      MOV     K1 U0\G4402
      MOV     K1 U0\G4502
      MOV     K1 U0\G4602
      MOV     K1 U0\G4702
      MOV     K1 U0\G4802
      MOV     K1 U0\G4902
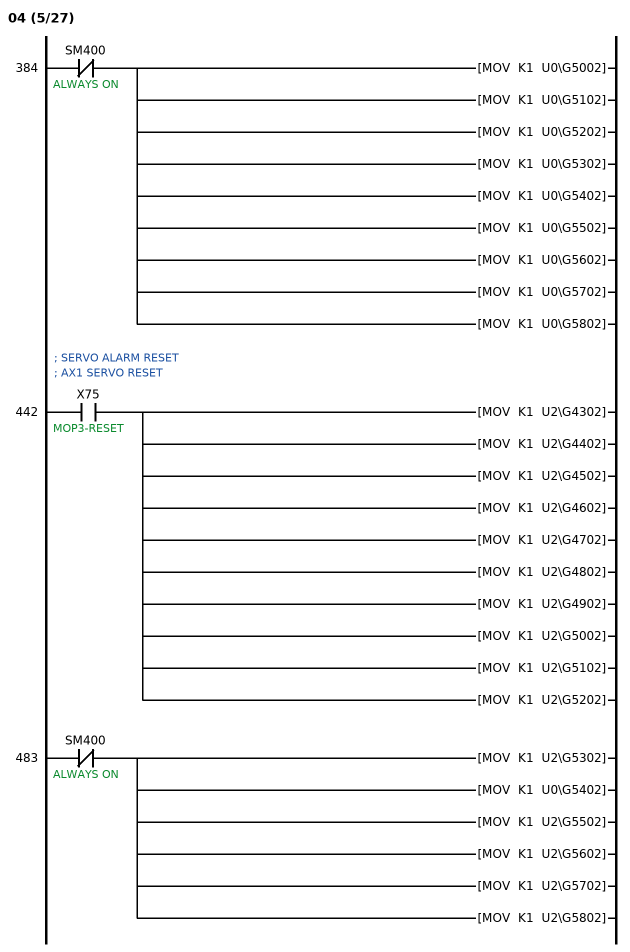
384   LDI     SM400  ; ALWAYS ON
      MOV     K1 U0\G5002
      MOV     K1 U0\G5102
      MOV     K1 U0\G5202
      MOV     K1 U0\G5302
      MOV     K1 U0\G5402
      MOV     K1 U0\G5502
      MOV     K1 U0\G5602
      MOV     K1 U0\G5702
      MOV     K1 U0\G5802
; SERVO ALARM RESET
; AX1 SERVO RESET
442   LD      X75  ; MOP3-RESET
      MOV     K1 U2\G4302
      MOV     K1 U2\G4402
      MOV     K1 U2\G4502
      MOV     K1 U2\G4602
      MOV     K1 U2\G4702
      MOV     K1 U2\G4802
      MOV     K1 U2\G4902
      MOV     K1 U2\G5002
      MOV     K1 U2\G5102
      MOV     K1 U2\G5202
483   LDI     SM400  ; ALWAYS ON
      MOV     K1 U2\G5302
      MOV     K1 U0\G5402
      MOV     K1 U2\G5502
      MOV     K1 U2\G5602
      MOV     K1 U2\G5702
      MOV     K1 U2\G5802
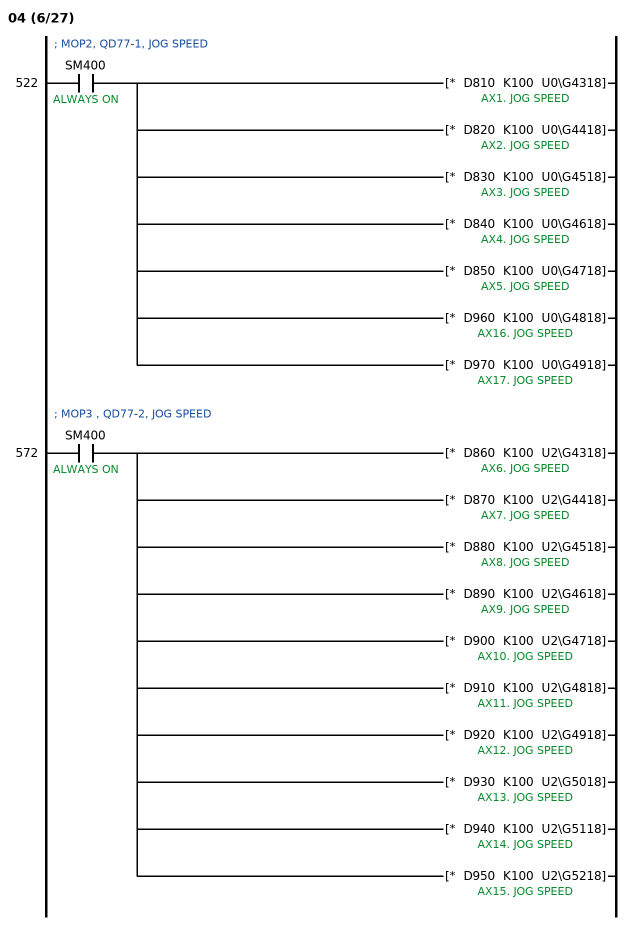
; MOP2, QD77-1, JOG SPEED
522   LD      SM400  ; ALWAYS ON
      *       D810 K100 U0\G4318  ; AX1. JOG SPEED
      *       D820 K100 U0\G4418  ; AX2. JOG SPEED
      *       D830 K100 U0\G4518  ; AX3. JOG SPEED
      *       D840 K100 U0\G4618  ; AX4. JOG SPEED
      *       D850 K100 U0\G4718  ; AX5. JOG SPEED
      *       D960 K100 U0\G4818  ; AX16. JOG SPEED
      *       D970 K100 U0\G4918  ; AX17. JOG SPEED
; MOP3 , QD77-2, JOG SPEED
572   LD      SM400  ; ALWAYS ON
      *       D860 K100 U2\G4318  ; AX6. JOG SPEED
      *       D870 K100 U2\G4418  ; AX7. JOG SPEED
      *       D880 K100 U2\G4518  ; AX8. JOG SPEED
      *       D890 K100 U2\G4618  ; AX9. JOG SPEED
      *       D900 K100 U2\G4718  ; AX10. JOG SPEED
      *       D910 K100 U2\G4818  ; AX11. JOG SPEED
      *       D920 K100 U2\G4918  ; AX12. JOG SPEED
      *       D930 K100 U2\G5018  ; AX13. JOG SPEED
      *       D940 K100 U2\G5118  ; AX14. JOG SPEED
      *       D950 K100 U2\G5218  ; AX15. JOG SPEED
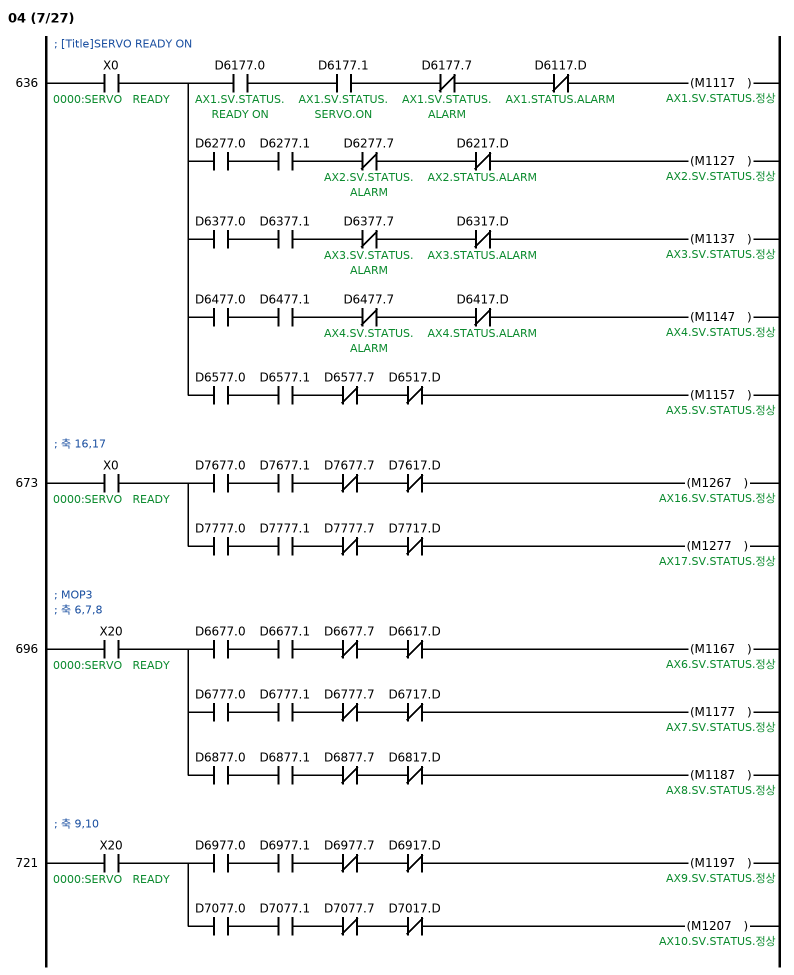
; [Title]SERVO READY ON
636   LD      X0  ; 0000:SERVO   READY
      MPS
      AND     D6177.0  ; AX1.SV.STATUS.READY ON
      AND     D6177.1  ; AX1.SV.STATUS.SERVO.ON
      ANI     D6177.7  ; AX1.SV.STATUS.ALARM
      ANI     D6117.D  ; AX1.STATUS.ALARM
      OUT     M1117  ; AX1.SV.STATUS.정상
      MRD
      AND     D6277.0
      AND     D6277.1
      ANI     D6277.7  ; AX2.SV.STATUS.ALARM
      ANI     D6217.D  ; AX2.STATUS.ALARM
      OUT     M1127  ; AX2.SV.STATUS.정상
      MRD
      AND     D6377.0
      AND     D6377.1
      ANI     D6377.7  ; AX3.SV.STATUS.ALARM
      ANI     D6317.D  ; AX3.STATUS.ALARM
      OUT     M1137  ; AX3.SV.STATUS.정상
      MRD
      AND     D6477.0
      AND     D6477.1
      ANI     D6477.7  ; AX4.SV.STATUS.ALARM
      ANI     D6417.D  ; AX4.STATUS.ALARM
      OUT     M1147  ; AX4.SV.STATUS.정상
      MPP
      AND     D6577.0
      AND     D6577.1
      ANI     D6577.7
      ANI     D6517.D
      OUT     M1157  ; AX5.SV.STATUS.정상
; 축 16,17
673   LD      X0  ; 0000:SERVO   READY
      MPS
      AND     D7677.0
      AND     D7677.1
      ANI     D7677.7
      ANI     D7617.D
      OUT     M1267  ; AX16.SV.STATUS.정상
      MPP
      AND     D7777.0
      AND     D7777.1
      ANI     D7777.7
      ANI     D7717.D
      OUT     M1277  ; AX17.SV.STATUS.정상
; MOP3
; 축 6,7,8
696   LD      X20  ; 0000:SERVO   READY
      MPS
      AND     D6677.0
      AND     D6677.1
      ANI     D6677.7
      ANI     D6617.D
      OUT     M1167  ; AX6.SV.STATUS.정상
      MRD
      AND     D6777.0
      AND     D6777.1
      ANI     D6777.7
      ANI     D6717.D
      OUT     M1177  ; AX7.SV.STATUS.정상
      MPP
      AND     D6877.0
      AND     D6877.1
      ANI     D6877.7
      ANI     D6817.D
      OUT     M1187  ; AX8.SV.STATUS.정상
; 축 9,10
721   LD      X20  ; 0000:SERVO   READY
      MPS
      AND     D6977.0
      AND     D6977.1
      ANI     D6977.7
      ANI     D6917.D
      OUT     M1197  ; AX9.SV.STATUS.정상
      MPP
      AND     D7077.0
      AND     D7077.1
      ANI     D7077.7
      ANI     D7017.D
      OUT     M1207  ; AX10.SV.STATUS.정상
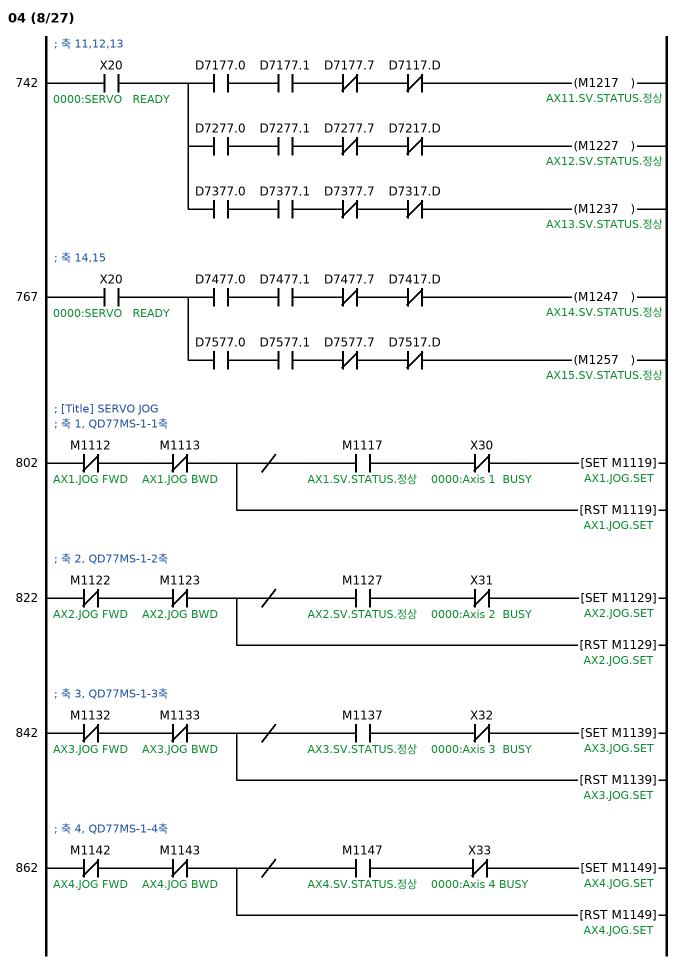
; 축 11,12,13
742   LD      X20  ; 0000:SERVO   READY
      MPS
      AND     D7177.0
      AND     D7177.1
      ANI     D7177.7
      ANI     D7117.D
      OUT     M1217  ; AX11.SV.STATUS.정상
      MRD
      AND     D7277.0
      AND     D7277.1
      ANI     D7277.7
      ANI     D7217.D
      OUT     M1227  ; AX12.SV.STATUS.정상
      MPP
      AND     D7377.0
      AND     D7377.1
      ANI     D7377.7
      ANI     D7317.D
      OUT     M1237  ; AX13.SV.STATUS.정상
; 축 14,15
767   LD      X20  ; 0000:SERVO   READY
      MPS
      AND     D7477.0
      AND     D7477.1
      ANI     D7477.7
      ANI     D7417.D
      OUT     M1247  ; AX14.SV.STATUS.정상
      MPP
      AND     D7577.0
      AND     D7577.1
      ANI     D7577.7
      ANI     D7517.D
      OUT     M1257  ; AX15.SV.STATUS.정상
; [Title] SERVO JOG
; 축 1, QD77MS-1-1축
802   LDI     M1112  ; AX1.JOG FWD
      ANI     M1113  ; AX1.JOG BWD
      MPS
      INV
      AND     M1117  ; AX1.SV.STATUS.정상
      ANI     X30  ; 0000:Axis 1  BUSY
      SET     M1119  ; AX1.JOG.SET
      MPP
      RST     M1119  ; AX1.JOG.SET
; 축 2, QD77MS-1-2축
822   LDI     M1122  ; AX2.JOG FWD
      ANI     M1123  ; AX2.JOG BWD
      MPS
      INV
      AND     M1127  ; AX2.SV.STATUS.정상
      ANI     X31  ; 0000:Axis 2  BUSY
      SET     M1129  ; AX2.JOG.SET
      MPP
      RST     M1129  ; AX2.JOG.SET
; 축 3, QD77MS-1-3축
842   LDI     M1132  ; AX3.JOG FWD
      ANI     M1133  ; AX3.JOG BWD
      MPS
      INV
      AND     M1137  ; AX3.SV.STATUS.정상
      ANI     X32  ; 0000:Axis 3  BUSY
      SET     M1139  ; AX3.JOG.SET
      MPP
      RST     M1139  ; AX3.JOG.SET
; 축 4, QD77MS-1-4축
862   LDI     M1142  ; AX4.JOG FWD
      ANI     M1143  ; AX4.JOG BWD
      MPS
      INV
      AND     M1147  ; AX4.SV.STATUS.정상
      ANI     X33  ; 0000:Axis 4 BUSY
      SET     M1149  ; AX4.JOG.SET
      MPP
      RST     M1149  ; AX4.JOG.SET
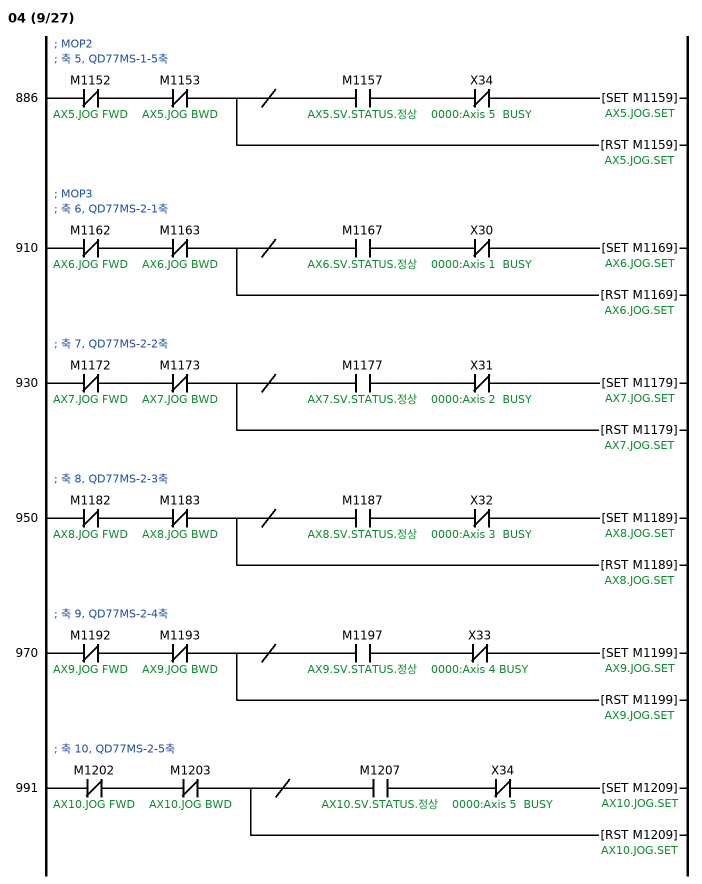
; MOP2
; 축 5, QD77MS-1-5축
886   LDI     M1152  ; AX5.JOG FWD
      ANI     M1153  ; AX5.JOG BWD
      MPS
      INV
      AND     M1157  ; AX5.SV.STATUS.정상
      ANI     X34  ; 0000:Axis 5  BUSY
      SET     M1159  ; AX5.JOG.SET
      MPP
      RST     M1159  ; AX5.JOG.SET
; MOP3
; 축 6, QD77MS-2-1축
910   LDI     M1162  ; AX6.JOG FWD
      ANI     M1163  ; AX6.JOG BWD
      MPS
      INV
      AND     M1167  ; AX6.SV.STATUS.정상
      ANI     X30  ; 0000:Axis 1  BUSY
      SET     M1169  ; AX6.JOG.SET
      MPP
      RST     M1169  ; AX6.JOG.SET
; 축 7, QD77MS-2-2축
930   LDI     M1172  ; AX7.JOG FWD
      ANI     M1173  ; AX7.JOG BWD
      MPS
      INV
      AND     M1177  ; AX7.SV.STATUS.정상
      ANI     X31  ; 0000:Axis 2  BUSY
      SET     M1179  ; AX7.JOG.SET
      MPP
      RST     M1179  ; AX7.JOG.SET
; 축 8, QD77MS-2-3축
950   LDI     M1182  ; AX8.JOG FWD
      ANI     M1183  ; AX8.JOG BWD
      MPS
      INV
      AND     M1187  ; AX8.SV.STATUS.정상
      ANI     X32  ; 0000:Axis 3  BUSY
      SET     M1189  ; AX8.JOG.SET
      MPP
      RST     M1189  ; AX8.JOG.SET
; 축 9, QD77MS-2-4축
970   LDI     M1192  ; AX9.JOG FWD
      ANI     M1193  ; AX9.JOG BWD
      MPS
      INV
      AND     M1197  ; AX9.SV.STATUS.정상
      ANI     X33  ; 0000:Axis 4 BUSY
      SET     M1199  ; AX9.JOG.SET
      MPP
      RST     M1199  ; AX9.JOG.SET
; 축 10, QD77MS-2-5축
991   LDI     M1202  ; AX10.JOG FWD
      ANI     M1203  ; AX10.JOG BWD
      MPS
      INV
      AND     M1207  ; AX10.SV.STATUS.정상
      ANI     X34  ; 0000:Axis 5  BUSY
      SET     M1209  ; AX10.JOG.SET
      MPP
      RST     M1209  ; AX10.JOG.SET
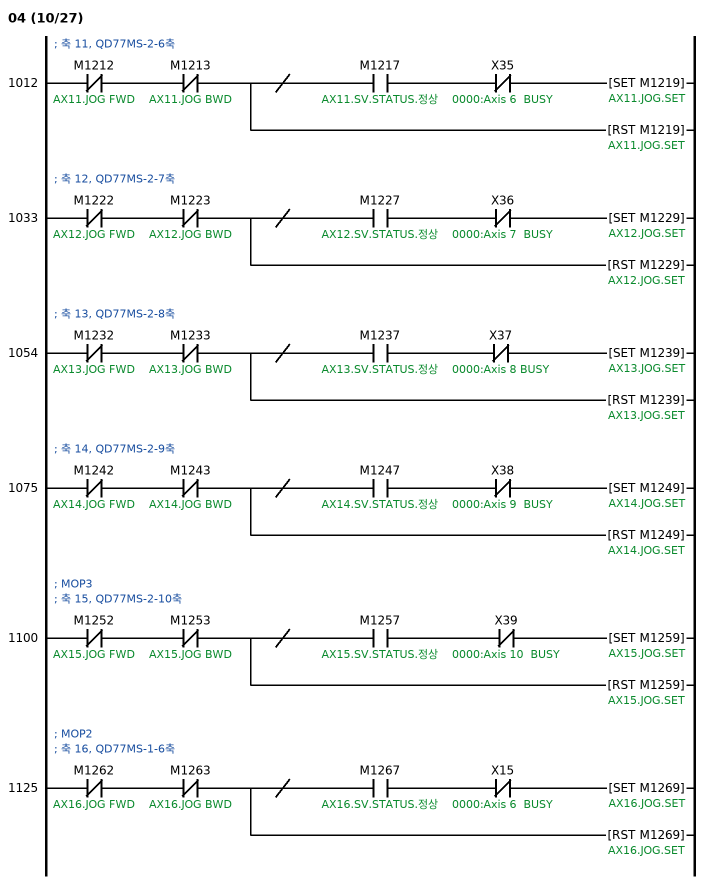
; 축 11, QD77MS-2-6축
1012  LDI     M1212  ; AX11.JOG FWD
      ANI     M1213  ; AX11.JOG BWD
      MPS
      INV
      AND     M1217  ; AX11.SV.STATUS.정상
      ANI     X35  ; 0000:Axis 6  BUSY
      SET     M1219  ; AX11.JOG.SET
      MPP
      RST     M1219  ; AX11.JOG.SET
; 축 12, QD77MS-2-7축
1033  LDI     M1222  ; AX12.JOG FWD
      ANI     M1223  ; AX12.JOG BWD
      MPS
      INV
      AND     M1227  ; AX12.SV.STATUS.정상
      ANI     X36  ; 0000:Axis 7  BUSY
      SET     M1229  ; AX12.JOG.SET
      MPP
      RST     M1229  ; AX12.JOG.SET
; 축 13, QD77MS-2-8축
1054  LDI     M1232  ; AX13.JOG FWD
      ANI     M1233  ; AX13.JOG BWD
      MPS
      INV
      AND     M1237  ; AX13.SV.STATUS.정상
      ANI     X37  ; 0000:Axis 8 BUSY
      SET     M1239  ; AX13.JOG.SET
      MPP
      RST     M1239  ; AX13.JOG.SET
; 축 14, QD77MS-2-9축
1075  LDI     M1242  ; AX14.JOG FWD
      ANI     M1243  ; AX14.JOG BWD
      MPS
      INV
      AND     M1247  ; AX14.SV.STATUS.정상
      ANI     X38  ; 0000:Axis 9  BUSY
      SET     M1249  ; AX14.JOG.SET
      MPP
      RST     M1249  ; AX14.JOG.SET
; MOP3
; 축 15, QD77MS-2-10축
1100  LDI     M1252  ; AX15.JOG FWD
      ANI     M1253  ; AX15.JOG BWD
      MPS
      INV
      AND     M1257  ; AX15.SV.STATUS.정상
      ANI     X39  ; 0000:Axis 10  BUSY
      SET     M1259  ; AX15.JOG.SET
      MPP
      RST     M1259  ; AX15.JOG.SET
; MOP2
; 축 16, QD77MS-1-6축
1125  LDI     M1262  ; AX16.JOG FWD
      ANI     M1263  ; AX16.JOG BWD
      MPS
      INV
      AND     M1267  ; AX16.SV.STATUS.정상
      ANI     X15  ; 0000:Axis 6  BUSY
      SET     M1269  ; AX16.JOG.SET
      MPP
      RST     M1269  ; AX16.JOG.SET
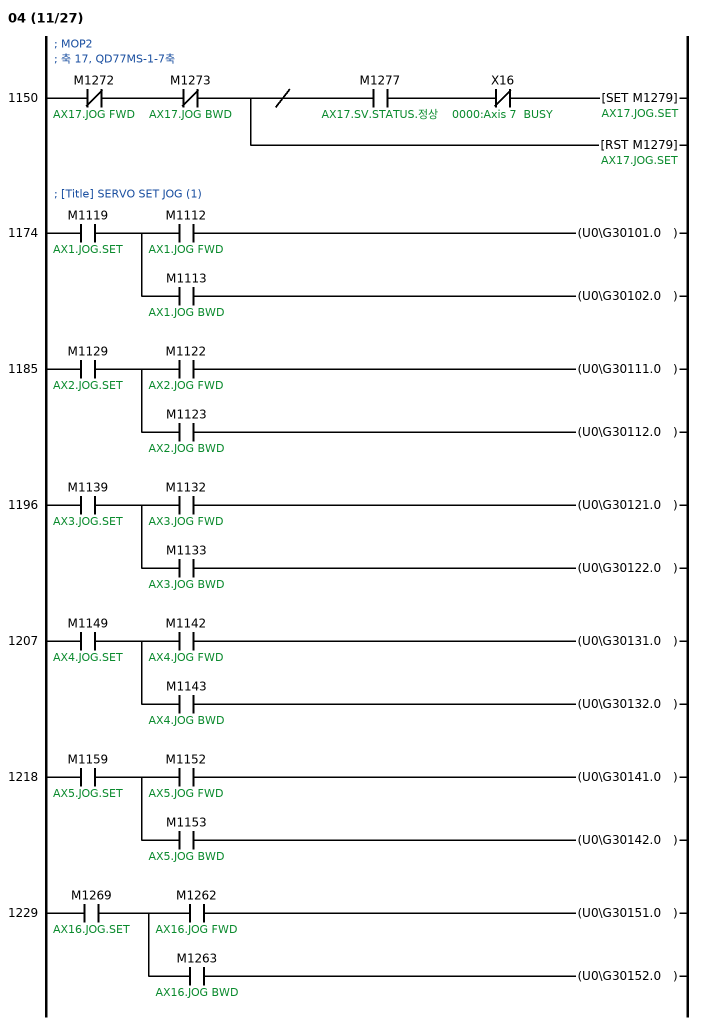
; MOP2
; 축 17, QD77MS-1-7축
1150  LDI     M1272  ; AX17.JOG FWD
      ANI     M1273  ; AX17.JOG BWD
      MPS
      INV
      AND     M1277  ; AX17.SV.STATUS.정상
      ANI     X16  ; 0000:Axis 7  BUSY
      SET     M1279  ; AX17.JOG.SET
      MPP
      RST     M1279  ; AX17.JOG.SET
; [Title] SERVO SET JOG (1)
1174  LD      M1119  ; AX1.JOG.SET
      MPS
      AND     M1112  ; AX1.JOG FWD
      OUT     U0\G30101.0
      MPP
      AND     M1113  ; AX1.JOG BWD
      OUT     U0\G30102.0
1185  LD      M1129  ; AX2.JOG.SET
      MPS
      AND     M1122  ; AX2.JOG FWD
      OUT     U0\G30111.0
      MPP
      AND     M1123  ; AX2.JOG BWD
      OUT     U0\G30112.0
1196  LD      M1139  ; AX3.JOG.SET
      MPS
      AND     M1132  ; AX3.JOG FWD
      OUT     U0\G30121.0
      MPP
      AND     M1133  ; AX3.JOG BWD
      OUT     U0\G30122.0
1207  LD      M1149  ; AX4.JOG.SET
      MPS
      AND     M1142  ; AX4.JOG FWD
      OUT     U0\G30131.0
      MPP
      AND     M1143  ; AX4.JOG BWD
      OUT     U0\G30132.0
1218  LD      M1159  ; AX5.JOG.SET
      MPS
      AND     M1152  ; AX5.JOG FWD
      OUT     U0\G30141.0
      MPP
      AND     M1153  ; AX5.JOG BWD
      OUT     U0\G30142.0
1229  LD      M1269  ; AX16.JOG.SET
      MPS
      AND     M1262  ; AX16.JOG FWD
      OUT     U0\G30151.0
      MPP
      AND     M1263  ; AX16.JOG BWD
      OUT     U0\G30152.0
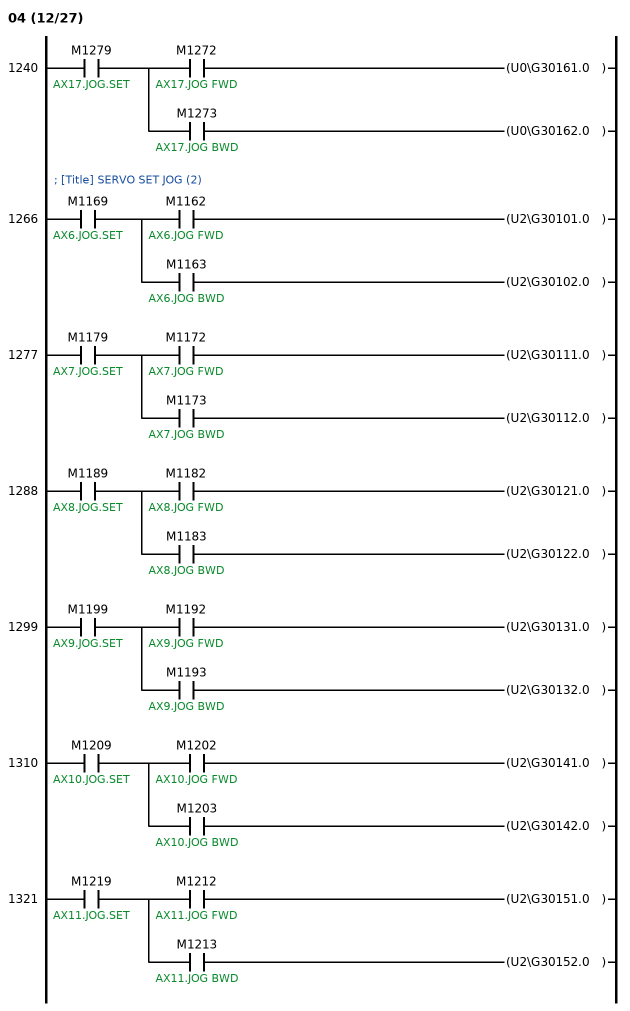
1240  LD      M1279  ; AX17.JOG.SET
      MPS
      AND     M1272  ; AX17.JOG FWD
      OUT     U0\G30161.0
      MPP
      AND     M1273  ; AX17.JOG BWD
      OUT     U0\G30162.0
; [Title] SERVO SET JOG (2)
1266  LD      M1169  ; AX6.JOG.SET
      MPS
      AND     M1162  ; AX6.JOG FWD
      OUT     U2\G30101.0
      MPP
      AND     M1163  ; AX6.JOG BWD
      OUT     U2\G30102.0
1277  LD      M1179  ; AX7.JOG.SET
      MPS
      AND     M1172  ; AX7.JOG FWD
      OUT     U2\G30111.0
      MPP
      AND     M1173  ; AX7.JOG BWD
      OUT     U2\G30112.0
1288  LD      M1189  ; AX8.JOG.SET
      MPS
      AND     M1182  ; AX8.JOG FWD
      OUT     U2\G30121.0
      MPP
      AND     M1183  ; AX8.JOG BWD
      OUT     U2\G30122.0
1299  LD      M1199  ; AX9.JOG.SET
      MPS
      AND     M1192  ; AX9.JOG FWD
      OUT     U2\G30131.0
      MPP
      AND     M1193  ; AX9.JOG BWD
      OUT     U2\G30132.0
1310  LD      M1209  ; AX10.JOG.SET
      MPS
      AND     M1202  ; AX10.JOG FWD
      OUT     U2\G30141.0
      MPP
      AND     M1203  ; AX10.JOG BWD
      OUT     U2\G30142.0
1321  LD      M1219  ; AX11.JOG.SET
      MPS
      AND     M1212  ; AX11.JOG FWD
      OUT     U2\G30151.0
      MPP
      AND     M1213  ; AX11.JOG BWD
      OUT     U2\G30152.0
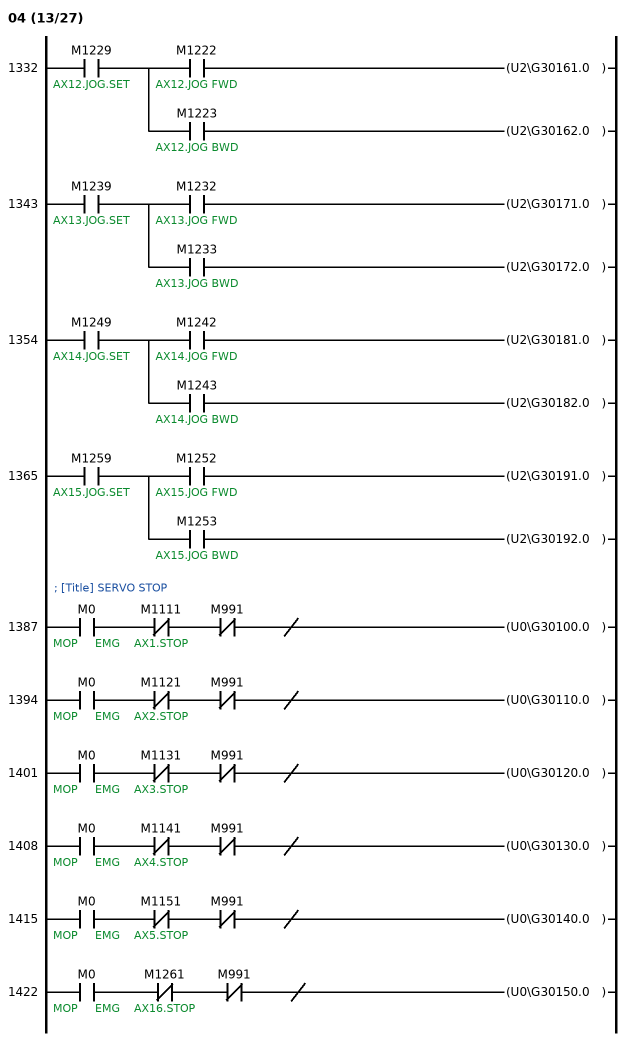
1332  LD      M1229  ; AX12.JOG.SET
      MPS
      AND     M1222  ; AX12.JOG FWD
      OUT     U2\G30161.0
      MPP
      AND     M1223  ; AX12.JOG BWD
      OUT     U2\G30162.0
1343  LD      M1239  ; AX13.JOG.SET
      MPS
      AND     M1232  ; AX13.JOG FWD
      OUT     U2\G30171.0
      MPP
      AND     M1233  ; AX13.JOG BWD
      OUT     U2\G30172.0
1354  LD      M1249  ; AX14.JOG.SET
      MPS
      AND     M1242  ; AX14.JOG FWD
      OUT     U2\G30181.0
      MPP
      AND     M1243  ; AX14.JOG BWD
      OUT     U2\G30182.0
1365  LD      M1259  ; AX15.JOG.SET
      MPS
      AND     M1252  ; AX15.JOG FWD
      OUT     U2\G30191.0
      MPP
      AND     M1253  ; AX15.JOG BWD
      OUT     U2\G30192.0
; [Title] SERVO STOP
1387  LD      M0  ; MOP     EMG
      ANI     M1111  ; AX1.STOP
      ANI     M991
      INV
      OUT     U0\G30100.0
1394  LD      M0  ; MOP     EMG
      ANI     M1121  ; AX2.STOP
      ANI     M991
      INV
      OUT     U0\G30110.0
1401  LD      M0  ; MOP     EMG
      ANI     M1131  ; AX3.STOP
      ANI     M991
      INV
      OUT     U0\G30120.0
1408  LD      M0  ; MOP     EMG
      ANI     M1141  ; AX4.STOP
      ANI     M991
      INV
      OUT     U0\G30130.0
1415  LD      M0  ; MOP     EMG
      ANI     M1151  ; AX5.STOP
      ANI     M991
      INV
      OUT     U0\G30140.0
1422  LD      M0  ; MOP     EMG
      ANI     M1261  ; AX16.STOP
      ANI     M991
      INV
      OUT     U0\G30150.0
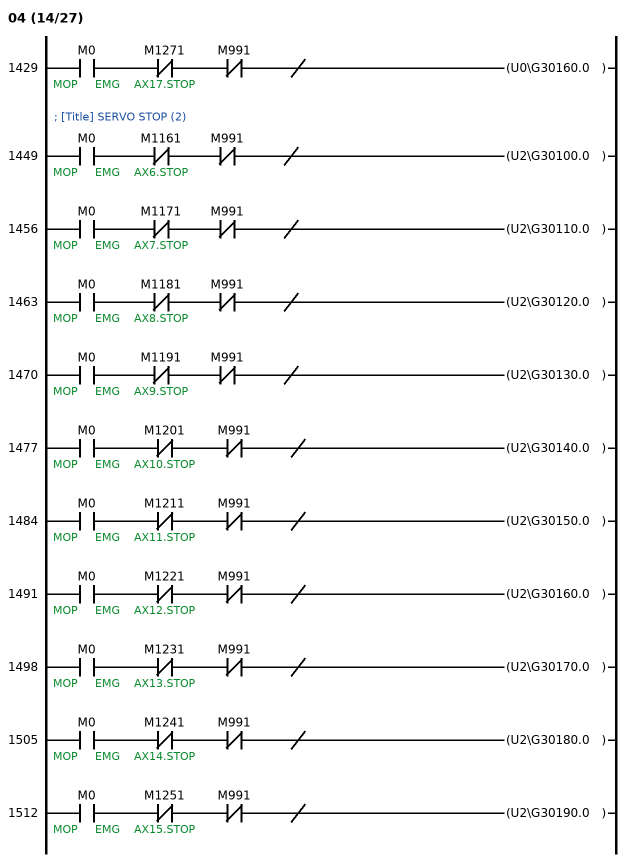
1429  LD      M0  ; MOP     EMG
      ANI     M1271  ; AX17.STOP
      ANI     M991
      INV
      OUT     U0\G30160.0
; [Title] SERVO STOP (2)
1449  LD      M0  ; MOP     EMG
      ANI     M1161  ; AX6.STOP
      ANI     M991
      INV
      OUT     U2\G30100.0
1456  LD      M0  ; MOP     EMG
      ANI     M1171  ; AX7.STOP
      ANI     M991
      INV
      OUT     U2\G30110.0
1463  LD      M0  ; MOP     EMG
      ANI     M1181  ; AX8.STOP
      ANI     M991
      INV
      OUT     U2\G30120.0
1470  LD      M0  ; MOP     EMG
      ANI     M1191  ; AX9.STOP
      ANI     M991
      INV
      OUT     U2\G30130.0
1477  LD      M0  ; MOP     EMG
      ANI     M1201  ; AX10.STOP
      ANI     M991
      INV
      OUT     U2\G30140.0
1484  LD      M0  ; MOP     EMG
      ANI     M1211  ; AX11.STOP
      ANI     M991
      INV
      OUT     U2\G30150.0
1491  LD      M0  ; MOP     EMG
      ANI     M1221  ; AX12.STOP
      ANI     M991
      INV
      OUT     U2\G30160.0
1498  LD      M0  ; MOP     EMG
      ANI     M1231  ; AX13.STOP
      ANI     M991
      INV
      OUT     U2\G30170.0
1505  LD      M0  ; MOP     EMG
      ANI     M1241  ; AX14.STOP
      ANI     M991
      INV
      OUT     U2\G30180.0
1512  LD      M0  ; MOP     EMG
      ANI     M1251  ; AX15.STOP
      ANI     M991
      INV
      OUT     U2\G30190.0
